LIN {X -0.145,Y -419.062,Z 861.894,A 0.000,B 0.000,C 90.000,E1 196.913} C_DIS
LIN {X 0.067,Y -417.772,Z 861.890,A 0.000,B 0.000,C 90.000,E1 196.205} C_DIS
LIN {X -0.189,Y -414.230,Z 861.881,A 0.000,B 0.000,C 90.000,E1 194.537} C_DIS
LIN {X -0.049,Y -408.722,Z 861.865,A 0.000,B 0.000,C 90.000,E1 191.771} C_DIS
LIN {X 0.119,Y -405.418,Z 861.856,A 0.000,B 0.000,C 90.000,E1 190.018} C_DIS
LIN {X 0.145,Y -402.699,Z 861.848,A 0.000,B 0.000,C 90.000,E1 188.624} C_DIS
LIN {X -0.116,Y -396.599,Z 861.831,A 0.000,B 0.000,C 90.000,E1 185.511} C_DIS
LIN {X -0.014,Y -390.296,Z 861.809,A 0.000,B 0.000,C 90.000,E1 181.604} C_DIS
LIN {X -0.149,Y -387.352,Z 861.797,A 0.000,B 0.000,C 90.000,E1 179.484} C_DIS
LIN {X 0.143,Y -384.816,Z 861.787,A 0.000,B 0.000,C 90.000,E1 177.650} C_DIS
LIN {X 0.018,Y -382.276,Z 861.777,A 0.000,B 0.000,C 90.000,E1 175.869} C_DIS
LIN {X 0.023,Y -378.755,Z 861.763,A 0.000,B 0.000,C 90.000,E1 173.337} C_DIS
LIN {X -0.169,Y -374.046,Z 861.739,A 0.000,B 0.000,C 90.000,E1 168.993} C_DIS
LIN {X -0.121,Y -373.099,Z 861.731,A 0.000,B 0.000,C 90.000,E1 167.521} C_DIS
LIN {X 0.156,Y -372.522,Z 861.720,A 0.000,B 0.000,C 90.000,E1 165.644} C_DIS
LIN {X -0.047,Y -372.718,Z 861.714,A 0.000,B 0.000,C 90.000,E1 164.574} C_DIS
LIN {X -0.080,Y -373.031,Z 861.712,A 0.000,B 0.000,C 90.000,E1 164.212} C_DIS
LIN {X -0.112,Y -373.157,Z 861.710,A 0.000,B 0.000,C 90.000,E1 163.850} C_DIS
LIN {X 0.127,Y -374.050,Z 861.705,A 0.000,B 0.000,C 90.000,E1 162.906} C_DIS
LIN {X 0.110,Y -375.461,Z 861.701,A 0.000,B 0.000,C 90.000,E1 162.127} C_DIS
LIN {X -0.174,Y -377.164,Z 861.698,A 0.000,B 0.000,C 90.000,E1 161.583} C_DIS
LIN {X -0.198,Y -379.423,Z 861.695,A 0.000,B 0.000,C 90.000,E1 161.040} C_DIS
LIN {X -0.203,Y -380.503,Z 861.694,A 0.000,B 0.000,C 90.000,E1 160.859} C_DIS
LIN {X -0.013,Y -383.679,Z 861.691,A 0.000,B 0.000,C 90.000,E1 160.369} C_DIS
LIN {X -0.012,Y -384.839,Z 861.690,A 0.000,B 0.000,C 90.000,E1 160.188} C_DIS
LIN {X -0.006,Y -386.584,Z 861.689,A 0.000,B 0.000,C 90.000,E1 160.007} C_DIS
LIN {X 0.011,Y -390.554,Z 861.687,A 0.000,B 0.000,C 90.000,E1 159.699} C_DIS
LIN {X 0.021,Y -392.446,Z 861.687,A 0.000,B 0.000,C 90.000,E1 159.571} C_DIS
LIN {X -0.042,Y -399.708,Z 861.685,A 0.000,B 0.000,C 90.000,E1 159.209} C_DIS
LIN {X -0.124,Y -407.378,Z 861.683,A 0.000,B 0.000,C 90.000,E1 158.901} C_DIS
LIN {X 0.178,Y -417.633,Z 861.680,A 0.000,B 0.000,C 90.000,E1 158.411} C_DIS
LIN {X -0.153,Y -425.580,Z 861.678,A 0.000,B 0.000,C 90.000,E1 158.028} C_DIS
LIN {X 0.034,Y -430.708,Z 861.676,A 0.000,B 0.000,C 90.000,E1 157.720} C_DIS
LIN {X -0.009,Y -433.655,Z 861.675,A 0.000,B 0.000,C 90.000,E1 157.539} C_DIS
LIN {X 0.068,Y -443.090,Z 861.672,A 0.000,B 0.000,C 90.000,E1 156.869} C_DIS
LIN {X -0.102,Y -447.734,Z 861.670,A 0.000,B 0.000,C 90.000,E1 156.538} C_DIS
LIN {X -0.139,Y -453.905,Z 861.667,A 0.000,B 0.000,C 90.000,E1 156.049} C_DIS
LIN {X -0.016,Y -464.227,Z 861.662,A 0.000,B 0.000,C 90.000,E1 155.101} C_DIS
LIN {X -0.106,Y -467.028,Z 861.660,A 0.000,B 0.000,C 90.000,E1 154.845} C_DIS
LIN {X -0.183,Y -472.623,Z 861.657,A 0.000,B 0.000,C 90.000,E1 154.280} C_DIS
LIN {X 0.095,Y -479.409,Z 861.653,A 0.000,B 0.000,C 90.000,E1 153.512} C_DIS
LIN {X 0.027,Y -483.253,Z 861.651,A 0.000,B 0.000,C 90.000,E1 153.076} C_DIS
LIN {X 0.252,Y -489.483,Z 861.646,A 0.000,B 0.000,C 90.000,E1 152.281} C_DIS
LIN {X 0.089,Y -495.170,Z 861.642,A 0.000,B 0.000,C 90.000,E1 151.591} C_DIS
LIN {X -0.181,Y -498.463,Z 861.640,A 0.000,B 0.000,C 90.000,E1 151.179} C_DIS
LIN {X -0.187,Y -503.200,Z 861.637,A 0.000,B 0.000,C 90.000,E1 150.589} C_DIS
LIN {X -0.265,Y -507.508,Z 861.633,A 0.000,B 0.000,C 90.000,E1 149.999} C_DIS
LIN {X -0.313,Y -511.672,Z 861.630,A 0.000,B 0.000,C 90.000,E1 149.410} C_DIS
LIN {X -0.155,Y -514.945,Z 861.627,A 0.000,B 0.000,C 90.000,E1 148.948} C_DIS
LIN {X 0.049,Y -520.575,Z 861.623,A 0.000,B 0.000,C 90.000,E1 148.043} C_DIS
LIN {X -0.231,Y -523.324,Z 861.620,A 0.000,B 0.000,C 90.000,E1 147.661} C_DIS
LIN {X -0.052,Y -527.781,Z 861.616,A 0.000,B 0.000,C 90.000,E1 146.914} C_DIS
LIN {X 0.019,Y -529.512,Z 861.615,A 0.000,B 0.000,C 90.000,E1 146.628} C_DIS
LIN {X 0.099,Y -536.054,Z 861.608,A 0.000,B 0.000,C 90.000,E1 145.468} C_DIS
LIN {X 0.120,Y -540.641,Z 861.604,A 0.000,B 0.000,C 90.000,E1 144.609} C_DIS
LIN {X -0.090,Y -546.662,Z 861.597,A 0.000,B 0.000,C 90.000,E1 143.497} C_DIS
LIN {X -0.202,Y -555.631,Z 861.588,A 0.000,B 0.000,C 90.000,E1 141.823} C_DIS
LIN {X -0.222,Y -563.196,Z 861.580,A 0.000,B 0.000,C 90.000,E1 140.436} C_DIS
LIN {X 0.135,Y -568.936,Z 861.574,A 0.000,B 0.000,C 90.000,E1 139.299} C_DIS
LIN {X -0.104,Y -573.699,Z 861.569,A 0.000,B 0.000,C 90.000,E1 138.366} C_DIS
LIN {X 0.017,Y -579.006,Z 861.563,A 0.000,B 0.000,C 90.000,E1 137.268} C_DIS
LIN {X 0.313,Y -585.693,Z 861.555,A 0.000,B 0.000,C 90.000,E1 135.891} C_DIS
LIN {X 0.022,Y -591.612,Z 861.548,A 0.000,B 0.000,C 90.000,E1 134.717} C_DIS
LIN {X -0.261,Y -595.300,Z 861.544,A 0.000,B 0.000,C 90.000,E1 133.947} C_DIS
LIN {X -0.093,Y -599.038,Z 861.540,A 0.000,B 0.000,C 90.000,E1 133.137} C_DIS
LIN {X -0.266,Y -605.015,Z 861.532,A 0.000,B 0.000,C 90.000,E1 131.838} C_DIS
LIN {X -0.150,Y -609.482,Z 861.527,A 0.000,B 0.000,C 90.000,E1 130.782} C_DIS
LIN {X -0.152,Y -614.771,Z 861.519,A 0.000,B 0.000,C 90.000,E1 129.483} C_DIS
LIN {X -0.294,Y -618.739,Z 861.514,A 0.000,B 0.000,C 90.000,E1 128.463} C_DIS
LIN {X -0.263,Y -625.196,Z 861.504,A 0.000,B 0.000,C 90.000,E1 126.664} C_DIS
LIN {X 0.239,Y -628.788,Z 861.498,A 0.000,B 0.000,C 90.000,E1 125.598} C_DIS
LIN {X -0.091,Y -631.992,Z 861.492,A 0.000,B 0.000,C 90.000,E1 124.612} C_DIS
LIN {X -0.242,Y -633.538,Z 861.490,A 0.000,B 0.000,C 90.000,E1 124.119} C_DIS
LIN {X 0.038,Y -636.798,Z 861.482,A 0.000,B 0.000,C 90.000,E1 122.832} C_DIS
LIN {X -0.046,Y -638.637,Z 861.478,A 0.000,B 0.000,C 90.000,E1 122.084} C_DIS
LIN {X 0.323,Y -641.263,Z 861.471,A 0.000,B 0.000,C 90.000,E1 120.797} C_DIS
LIN {X -0.157,Y -643.563,Z 861.464,A 0.000,B 0.000,C 90.000,E1 119.589} C_DIS
LIN {X -0.018,Y -644.146,Z 861.462,A 0.000,B 0.000,C 90.000,E1 119.077} C_DIS
LIN {X 0.130,Y -645.007,Z 861.459,A 0.000,B 0.000,C 90.000,E1 118.565} C_DIS
LIN {X -0.036,Y -646.885,Z 861.452,A 0.000,B 0.000,C 90.000,E1 117.334} C_DIS
LIN {X 0.136,Y -647.533,Z 861.449,A 0.000,B 0.000,C 90.000,E1 116.821} C_DIS
LIN {X 0.000,Y -648.671,Z 861.442,A 0.000,B 0.000,C 90.000,E1 115.591} C_DIS
LIN {X 0.090,Y -649.085,Z 861.437,A 0.000,B 0.000,C 90.000,E1 114.591} C_DIS
LIN {X 0.182,Y -649.129,Z 861.435,A 0.000,B 0.000,C 90.000,E1 114.335} C_DIS
LIN {X 0.363,Y -648.828,Z 861.433,A 0.000,B 0.000,C 90.000,E1 113.823} C_DIS
LIN {X 0.192,Y -648.419,Z 861.431,A 0.000,B 0.000,C 90.000,E1 113.590} C_DIS
LIN {X -0.229,Y -647.091,Z 861.428,A 0.000,B 0.000,C 90.000,E1 113.131} C_DIS
LIN {X -0.359,Y -644.836,Z 861.426,A 0.000,B 0.000,C 90.000,E1 112.770} C_DIS
LIN {X -0.320,Y -644.240,Z 861.426,A 0.000,B 0.000,C 90.000,E1 112.642} C_DIS
LIN {X -0.284,Y -643.376,Z 861.425,A 0.000,B 0.000,C 90.000,E1 112.514} C_DIS
LIN {X 0.377,Y -641.224,Z 861.424,A 0.000,B 0.000,C 90.000,E1 112.206} C_DIS
LIN {X 0.168,Y -640.004,Z 861.423,A 0.000,B 0.000,C 90.000,E1 112.099} C_DIS
LIN {X 0.207,Y -638.590,Z 861.422,A 0.000,B 0.000,C 90.000,E1 111.972} C_DIS
LIN {X 0.247,Y -636.605,Z 861.422,A 0.000,B 0.000,C 90.000,E1 111.844} C_DIS
LIN {X -0.279,Y -635.300,Z 861.421,A 0.000,B 0.000,C 90.000,E1 111.844} C_DIS
LIN {X -0.212,Y -631.962,Z 861.420,A 0.000,B 0.000,C 90.000,E1 111.589} C_DIS
LIN {X 0.146,Y -628.475,Z 861.419,A 0.000,B 0.000,C 90.000,E1 111.354} C_DIS
LIN {X -0.016,Y -623.661,Z 861.417,A 0.000,B 0.000,C 90.000,E1 111.099} C_DIS
LIN {X 0.310,Y -597.380,Z 861.410,A 0.000,B 0.000,C 90.000,E1 109.812} C_DIS
LIN {X 0.154,Y -589.216,Z 861.408,A 0.000,B 0.000,C 90.000,E1 109.450} C_DIS
LIN {X -0.233,Y -583.699,Z 861.407,A 0.000,B 0.000,C 90.000,E1 109.268} C_DIS
LIN {X 0.287,Y -580.083,Z 861.406,A 0.000,B 0.000,C 90.000,E1 109.087} C_DIS
LIN {X -0.189,Y -572.340,Z 861.405,A 0.000,B 0.000,C 90.000,E1 108.906} C_DIS
LIN {X 0.205,Y -566.390,Z 861.404,A 0.000,B 0.000,C 90.000,E1 108.671} C_DIS
LIN {X 0.035,Y -563.220,Z 861.403,A 0.000,B 0.000,C 90.000,E1 108.489} C_DIS
LIN {X -0.011,Y -562.426,Z 861.402,A 0.000,B 0.000,C 90.000,E1 108.417} C_DIS
LIN {X -0.223,Y -561.003,Z 861.401,A 0.000,B 0.000,C 90.000,E1 108.181} C_DIS
LIN {X -0.201,Y -559.978,Z 861.399,A 0.000,B 0.000,C 90.000,E1 107.764} C_DIS
LIN {X -0.142,Y -559.387,Z 861.395,A 0.000,B 0.000,C 90.000,E1 107.149} C_DIS
LIN {X 0.043,Y -559.497,Z 861.384,A 0.000,B 0.000,C 90.000,E1 105.190} C_DIS
LIN {X 0.130,Y -560.677,Z 861.369,A 0.000,B 0.000,C 90.000,E1 102.411} C_DIS
LIN {X 0.142,Y -562.134,Z 861.357,A 0.000,B 0.000,C 90.000,E1 100.197} C_DIS
LIN {X -0.122,Y -563.310,Z 861.348,A 0.000,B 0.000,C 90.000,E1 98.568} C_DIS
LIN {X -0.050,Y -564.232,Z 861.340,A 0.000,B 0.000,C 90.000,E1 97.182} C_DIS
LIN {X 0.038,Y -565.001,Z 861.332,A 0.000,B 0.000,C 90.000,E1 95.796} C_DIS
LIN {X -0.232,Y -565.860,Z 861.322,A 0.000,B 0.000,C 90.000,E1 93.898} C_DIS
LIN {X -0.213,Y -566.345,Z 861.314,A 0.000,B 0.000,C 90.000,E1 92.522} C_DIS
LIN {X -0.068,Y -566.780,Z 861.305,A 0.000,B 0.000,C 90.000,E1 90.859} C_DIS
LIN {X -0.042,Y -567.118,Z 861.297,A 0.000,B 0.000,C 90.000,E1 89.484} C_DIS
LIN {X 0.002,Y -567.427,Z 861.290,A 0.000,B 0.000,C 90.000,E1 88.108} C_DIS
LIN {X -0.278,Y -567.763,Z 861.279,A 0.000,B 0.000,C 90.000,E1 86.216} C_DIS
LIN {X -0.189,Y -567.981,Z 861.271,A 0.000,B 0.000,C 90.000,E1 84.837} C_DIS
LIN {X 0.240,Y -568.334,Z 861.261,A 0.000,B 0.000,C 90.000,E1 82.875} C_DIS
LIN {X -0.272,Y -568.959,Z 861.248,A 0.000,B 0.000,C 90.000,E1 80.735} C_DIS
LIN {X -0.027,Y -569.755,Z 861.236,A 0.000,B 0.000,C 90.000,E1 78.522} C_DIS
LIN {X 0.160,Y -570.549,Z 861.226,A 0.000,B 0.000,C 90.000,E1 76.589} C_DIS
LIN {X -0.066,Y -570.893,Z 861.220,A 0.000,B 0.000,C 90.000,E1 75.519} C_DIS
LIN {X 0.270,Y -571.198,Z 861.214,A 0.000,B 0.000,C 90.000,E1 74.393} C_DIS
LIN {X 0.057,Y -571.465,Z 861.207,A 0.000,B 0.000,C 90.000,E1 73.323} C_DIS
LIN {X 0.164,Y -571.700,Z 861.197,A 0.000,B 0.000,C 90.000,E1 71.402} C_DIS
LIN {X -0.087,Y -571.730,Z 861.186,A 0.000,B 0.000,C 90.000,E1 69.518} C_DIS
LIN {X 0.249,Y -571.730,Z 861.177,A 0.000,B 0.000,C 90.000,E1 67.847} C_DIS
LIN {X 0.063,Y -571.623,Z 861.168,A 0.000,B 0.000,C 90.000,E1 66.230} C_DIS
LIN {X 0.270,Y -571.464,Z 861.160,A 0.000,B 0.000,C 90.000,E1 64.845} C_DIS
LIN {X -0.212,Y -571.079,Z 861.151,A 0.000,B 0.000,C 90.000,E1 63.256} C_DIS
LIN {X 0.054,Y -570.536,Z 861.142,A 0.000,B 0.000,C 90.000,E1 61.591} C_DIS
LIN {X -0.078,Y -570.026,Z 861.136,A 0.000,B 0.000,C 90.000,E1 60.511} C_DIS
LIN {X 0.179,Y -569.623,Z 861.132,A 0.000,B 0.000,C 90.000,E1 59.665} C_DIS
LIN {X -0.133,Y -568.550,Z 861.124,A 0.000,B 0.000,C 90.000,E1 58.329} C_DIS
LIN {X -0.088,Y -567.894,Z 861.119,A 0.000,B 0.000,C 90.000,E1 57.502} C_DIS
LIN {X -0.356,Y -567.033,Z 861.115,A 0.000,B 0.000,C 90.000,E1 56.707} C_DIS
LIN {X -0.213,Y -565.644,Z 861.109,A 0.000,B 0.000,C 90.000,E1 55.595} C_DIS
LIN {X -0.199,Y -564.517,Z 861.104,A 0.000,B 0.000,C 90.000,E1 54.769} C_DIS
LIN {X 0.234,Y -562.850,Z 861.098,A 0.000,B 0.000,C 90.000,E1 53.623} C_DIS
LIN {X -0.141,Y -560.884,Z 861.092,A 0.000,B 0.000,C 90.000,E1 52.557} C_DIS
LIN {X 0.145,Y -559.235,Z 861.087,A 0.000,B 0.000,C 90.000,E1 51.698} C_DIS
LIN {X -0.113,Y -558.053,Z 861.084,A 0.000,B 0.000,C 90.000,E1 51.170} C_DIS
LIN {X -0.294,Y -555.992,Z 861.080,A 0.000,B 0.000,C 90.000,E1 50.356} C_DIS
LIN {X 0.284,Y -553.563,Z 861.075,A 0.000,B 0.000,C 90.000,E1 49.461} C_DIS
LIN {X 0.050,Y -550.841,Z 861.070,A 0.000,B 0.000,C 90.000,E1 48.647} C_DIS
LIN {X 0.106,Y -548.875,Z 861.067,A 0.000,B 0.000,C 90.000,E1 48.081} C_DIS
LIN {X 0.187,Y -545.568,Z 861.063,A 0.000,B 0.000,C 90.000,E1 47.229} C_DIS
LIN {X 0.036,Y -542.567,Z 861.059,A 0.000,B 0.000,C 90.000,E1 46.539} C_DIS
LIN {X 0.228,Y -539.269,Z 861.055,A 0.000,B 0.000,C 90.000,E1 45.810} C_DIS
LIN {X 0.022,Y -537.203,Z 861.052,A 0.000,B 0.000,C 90.000,E1 45.405} C_DIS
LIN {X 0.165,Y -533.249,Z 861.048,A 0.000,B 0.000,C 90.000,E1 44.676} C_DIS
LIN {X 0.101,Y -529.791,Z 861.045,A 0.000,B 0.000,C 90.000,E1 44.109} C_DIS
LIN {X 0.077,Y -526.153,Z 861.042,A 0.000,B 0.000,C 90.000,E1 43.542} C_DIS
LIN {X -0.042,Y -522.226,Z 861.039,A 0.000,B 0.000,C 90.000,E1 42.975} C_DIS
LIN {X 0.193,Y -517.988,Z 861.036,A 0.000,B 0.000,C 90.000,E1 42.366} C_DIS
LIN {X -0.331,Y -513.435,Z 861.032,A 0.000,B 0.000,C 90.000,E1 41.838} C_DIS
LIN {X 0.055,Y -509.906,Z 861.030,A 0.000,B 0.000,C 90.000,E1 41.353} C_DIS
LIN {X 0.067,Y -504.988,Z 861.027,A 0.000,B 0.000,C 90.000,E1 40.782} C_DIS
LIN {X -0.141,Y -500.047,Z 861.024,A 0.000,B 0.000,C 90.000,E1 40.253} C_DIS
LIN {X -0.038,Y -495.889,Z 861.021,A 0.000,B 0.000,C 90.000,E1 39.806} C_DIS
LIN {X -0.212,Y -490.304,Z 861.018,A 0.000,B 0.000,C 90.000,E1 39.277} C_DIS
LIN {X -0.153,Y -481.649,Z 861.014,A 0.000,B 0.000,C 90.000,E1 38.463} C_DIS
LIN {X 0.113,Y -470.949,Z 861.009,A 0.000,B 0.000,C 90.000,E1 37.523} C_DIS
LIN {X 0.015,Y -464.758,Z 861.006,A 0.000,B 0.000,C 90.000,E1 37.030} C_DIS
LIN {X -0.286,Y -452.263,Z 861.000,A 0.000,B 0.000,C 90.000,E1 36.091} C_DIS
LIN {X 0.081,Y -438.081,Z 860.994,A 0.000,B 0.000,C 90.000,E1 34.945} C_DIS
LIN {X 0.012,Y -419.665,Z 860.986,A 0.000,B 0.000,C 90.000,E1 33.452} C_DIS
LIN {X 0.029,Y -404.695,Z 860.978,A 0.000,B 0.000,C 90.000,E1 32.084} C_DIS
LIN {X -0.041,Y -399.160,Z 860.975,A 0.000,B 0.000,C 90.000,E1 31.514} C_DIS
LIN {X -0.019,Y -394.767,Z 860.972,A 0.000,B 0.000,C 90.000,E1 30.924} C_DIS
LIN {X 0.013,Y -393.080,Z 860.970,A 0.000,B 0.000,C 90.000,E1 30.590} C_DIS
LIN {X 0.017,Y -392.132,Z 860.969,A 0.000,B 0.000,C 90.000,E1 30.413} C_DIS
LIN {X -0.239,Y -390.569,Z 860.966,A 0.000,B 0.000,C 90.000,E1 29.873} C_DIS
LIN {X -0.005,Y -389.839,Z 860.961,A 0.000,B 0.000,C 90.000,E1 28.949} C_DIS
LIN {X 0.031,Y -389.754,Z 860.957,A 0.000,B 0.000,C 90.000,E1 28.231} C_DIS
LIN {X -0.106,Y -392.270,Z 860.935,A 0.000,B 0.000,C 90.000,E1 24.335} C_DIS
LIN {X 0.208,Y -395.035,Z 860.917,A 0.000,B 0.000,C 90.000,E1 21.099} C_DIS
LIN {X -0.081,Y -397.526,Z 860.904,A 0.000,B 0.000,C 90.000,E1 18.671} C_DIS
LIN {X -0.087,Y -399.530,Z 860.894,A 0.000,B 0.000,C 90.000,E1 16.913} C_DIS
LIN {X -0.136,Y -403.103,Z 860.878,A 0.000,B 0.000,C 90.000,E1 14.120} C_DIS
LIN {X 0.129,Y -407.132,Z 860.863,A 0.000,B 0.000,C 90.000,E1 11.299} C_DIS
LIN {X -0.138,Y -410.967,Z 860.849,A 0.000,B 0.000,C 90.000,E1 8.916} C_DIS
LIN {X 0.088,Y -416.322,Z 860.832,A 0.000,B 0.000,C 90.000,E1 5.796} C_DIS
LIN {X -0.144,Y -420.094,Z 860.821,A 0.000,B 0.000,C 90.000,E1 3.784} C_DIS
LIN {X 0.203,Y -425.720,Z 860.806,A 0.000,B 0.000,C 90.000,E1 1.031} C_DIS
LIN {X -0.199,Y -429.433,Z 860.797,A 0.000,B 0.000,C 90.000,E1 359.484} C_DIS
LIN {X -0.076,Y -435.036,Z 860.784,A 0.000,B 0.000,C 90.000,E1 357.135} C_DIS
LIN {X -0.040,Y -441.939,Z 860.769,A 0.000,B 0.000,C 90.000,E1 354.489} C_DIS
LIN {X -0.159,Y -444.717,Z 860.765,A 0.000,B 0.000,C 90.000,E1 353.685} C_DIS
LIN {X -0.185,Y -446.635,Z 860.763,A 0.000,B 0.000,C 90.000,E1 353.280} C_DIS
LIN {X -0.205,Y -451.971,Z 860.759,A 0.000,B 0.000,C 90.000,E1 352.648} C_DIS
LIN {X -0.058,Y -455.920,Z 860.758,A 0.000,B 0.000,C 90.000,E1 352.356} C_DIS
LIN {X 0.064,Y -462.281,Z 860.756,A 0.000,B 0.000,C 90.000,E1 352.008} C_DIS
LIN {X -0.177,Y -473.870,Z 860.753,A 0.000,B 0.000,C 90.000,E1 351.489} C_DIS
LIN {X -0.152,Y -480.634,Z 860.751,A 0.000,B 0.000,C 90.000,E1 351.141} C_DIS
LIN {X 0.231,Y -486.952,Z 860.749,A 0.000,B 0.000,C 90.000,E1 350.735} C_DIS
LIN {X 0.226,Y -496.803,Z 860.745,A 0.000,B 0.000,C 90.000,E1 350.151} C_DIS
LIN {X 0.094,Y -507.807,Z 860.742,A 0.000,B 0.000,C 90.000,E1 349.454} C_DIS
LIN {X 0.192,Y -517.208,Z 860.738,A 0.000,B 0.000,C 90.000,E1 348.814} C_DIS
LIN {X 0.075,Y -526.384,Z 860.734,A 0.000,B 0.000,C 90.000,E1 348.173} C_DIS
LIN {X -0.235,Y -533.792,Z 860.731,A 0.000,B 0.000,C 90.000,E1 347.645} C_DIS
LIN {X -0.178,Y -541.052,Z 860.728,A 0.000,B 0.000,C 90.000,E1 347.048} C_DIS
LIN {X 0.009,Y -550.870,Z 860.723,A 0.000,B 0.000,C 90.000,E1 346.172} C_DIS
LIN {X -0.115,Y -560.007,Z 860.718,A 0.000,B 0.000,C 90.000,E1 345.283} C_DIS
LIN {X -0.172,Y -565.040,Z 860.715,A 0.000,B 0.000,C 90.000,E1 344.755} C_DIS
LIN {X 0.126,Y -572.253,Z 860.711,A 0.000,B 0.000,C 90.000,E1 343.921} C_DIS
LIN {X -0.148,Y -577.732,Z 860.707,A 0.000,B 0.000,C 90.000,E1 343.268} C_DIS
LIN {X 0.259,Y -583.987,Z 860.703,A 0.000,B 0.000,C 90.000,E1 342.417} C_DIS
LIN {X 0.146,Y -587.838,Z 860.700,A 0.000,B 0.000,C 90.000,E1 341.891} C_DIS
LIN {X 0.174,Y -592.324,Z 860.696,A 0.000,B 0.000,C 90.000,E1 341.221} C_DIS
LIN {X 0.189,Y -597.396,Z 860.691,A 0.000,B 0.000,C 90.000,E1 340.423} C_DIS
LIN {X 0.009,Y -602.864,Z 860.686,A 0.000,B 0.000,C 90.000,E1 339.518} C_DIS
LIN {X 0.047,Y -609.460,Z 860.680,A 0.000,B 0.000,C 90.000,E1 338.337} C_DIS
LIN {X 0.227,Y -614.416,Z 860.675,A 0.000,B 0.000,C 90.000,E1 337.411} C_DIS
LIN {X -0.111,Y -619.731,Z 860.669,A 0.000,B 0.000,C 90.000,E1 336.410} C_DIS
LIN {X 0.184,Y -623.516,Z 860.665,A 0.000,B 0.000,C 90.000,E1 335.613} C_DIS
LIN {X 0.233,Y -629.342,Z 860.658,A 0.000,B 0.000,C 90.000,E1 334.332} C_DIS
LIN {X 0.034,Y -632.552,Z 860.653,A 0.000,B 0.000,C 90.000,E1 333.589} C_DIS
LIN {X 0.141,Y -635.611,Z 860.649,A 0.000,B 0.000,C 90.000,E1 332.820} C_DIS
LIN {X -0.236,Y -639.523,Z 860.644,A 0.000,B 0.000,C 90.000,E1 331.847} C_DIS
LIN {X 0.310,Y -643.100,Z 860.638,A 0.000,B 0.000,C 90.000,E1 330.795} C_DIS
LIN {X 0.353,Y -646.615,Z 860.632,A 0.000,B 0.000,C 90.000,E1 329.793} C_DIS
LIN {X 0.030,Y -649.075,Z 860.628,A 0.000,B 0.000,C 90.000,E1 329.076} C_DIS
LIN {X -0.318,Y -652.863,Z 860.621,A 0.000,B 0.000,C 90.000,E1 327.867} C_DIS
LIN {X 0.201,Y -655.609,Z 860.616,A 0.000,B 0.000,C 90.000,E1 326.834} C_DIS
LIN {X 0.299,Y -657.575,Z 860.612,A 0.000,B 0.000,C 90.000,E1 326.087} C_DIS
LIN {X -0.100,Y -660.554,Z 860.605,A 0.000,B 0.000,C 90.000,E1 324.895} C_DIS
LIN {X -0.016,Y -662.610,Z 860.600,A 0.000,B 0.000,C 90.000,E1 323.909} C_DIS
LIN {X 0.092,Y -664.473,Z 860.594,A 0.000,B 0.000,C 90.000,E1 322.924} C_DIS
LIN {X 0.189,Y -666.414,Z 860.587,A 0.000,B 0.000,C 90.000,E1 321.698} C_DIS
LIN {X -0.205,Y -668.169,Z 860.581,A 0.000,B 0.000,C 90.000,E1 320.517} C_DIS
LIN {X 0.291,Y -669.078,Z 860.577,A 0.000,B 0.000,C 90.000,E1 319.747} C_DIS
LIN {X -0.061,Y -670.675,Z 860.568,A 0.000,B 0.000,C 90.000,E1 318.324} C_DIS
LIN {X 0.088,Y -672.973,Z 860.558,A 0.000,B 0.000,C 90.000,E1 316.377} C_DIS
LIN {X 0.201,Y -674.442,Z 860.551,A 0.000,B 0.000,C 90.000,E1 315.162} C_DIS
LIN {X 0.226,Y -674.593,Z 860.550,A 0.000,B 0.000,C 90.000,E1 314.919} C_DIS
LIN {X 0.253,Y -674.941,Z 860.548,A 0.000,B 0.000,C 90.000,E1 314.676} C_DIS
LIN {X 0.054,Y -677.032,Z 860.536,A 0.000,B 0.000,C 90.000,E1 312.528} C_DIS
LIN {X 0.265,Y -678.191,Z 860.530,A 0.000,B 0.000,C 90.000,E1 311.310} C_DIS
LIN {X 0.121,Y -679.752,Z 860.520,A 0.000,B 0.000,C 90.000,E1 309.644} C_DIS
LIN {X -0.091,Y -680.568,Z 860.515,A 0.000,B 0.000,C 90.000,E1 308.705} C_DIS
LIN {X -0.083,Y -681.939,Z 860.506,A 0.000,B 0.000,C 90.000,E1 307.030} C_DIS
LIN {X -0.078,Y -683.066,Z 860.498,A 0.000,B 0.000,C 90.000,E1 305.598} C_DIS
LIN {X -0.457,Y -684.012,Z 860.490,A 0.000,B 0.000,C 90.000,E1 304.199} C_DIS
LIN {X -0.060,Y -685.313,Z 860.479,A 0.000,B 0.000,C 90.000,E1 302.260} C_DIS
LIN {X 0.003,Y -686.563,Z 860.470,A 0.000,B 0.000,C 90.000,E1 300.590} C_DIS
LIN {X -0.245,Y -687.943,Z 860.461,A 0.000,B 0.000,C 90.000,E1 298.949} C_DIS
LIN {X -0.087,Y -689.285,Z 860.453,A 0.000,B 0.000,C 90.000,E1 297.513} C_DIS
LIN {X 0.016,Y -690.960,Z 860.444,A 0.000,B 0.000,C 90.000,E1 295.848} C_DIS
LIN {X 0.292,Y -692.132,Z 860.437,A 0.000,B 0.000,C 90.000,E1 294.643} C_DIS
LIN {X 0.099,Y -692.644,Z 860.433,A 0.000,B 0.000,C 90.000,E1 293.951} C_DIS
LIN {X -0.092,Y -692.634,Z 860.429,A 0.000,B 0.000,C 90.000,E1 293.259} C_DIS
LIN {X 0.114,Y -691.666,Z 860.427,A 0.000,B 0.000,C 90.000,E1 292.770} C_DIS
LIN {X 0.351,Y -690.965,Z 860.425,A 0.000,B 0.000,C 90.000,E1 292.514} C_DIS
LIN {X 0.203,Y -690.295,Z 860.425,A 0.000,B 0.000,C 90.000,E1 292.408} C_DIS
LIN {X -0.238,Y -686.592,Z 860.422,A 0.000,B 0.000,C 90.000,E1 291.972} C_DIS
LIN {X -0.127,Y -685.449,Z 860.421,A 0.000,B 0.000,C 90.000,E1 291.844} C_DIS
LIN {X -0.021,Y -683.688,Z 860.421,A 0.000,B 0.000,C 90.000,E1 291.716} C_DIS
LIN {X -0.179,Y -679.497,Z 860.420,A 0.000,B 0.000,C 90.000,E1 291.535} C_DIS
LIN {X 0.264,Y -676.010,Z 860.419,A 0.000,B 0.000,C 90.000,E1 291.354} C_DIS
LIN {X 0.166,Y -670.319,Z 860.418,A 0.000,B 0.000,C 90.000,E1 291.173} C_DIS
LIN {X 0.140,Y -656.825,Z 860.416,A 0.000,B 0.000,C 90.000,E1 290.865} C_DIS
LIN {X -0.130,Y -653.809,Z 860.415,A 0.000,B 0.000,C 90.000,E1 290.791} C_DIS
LIN {X -0.178,Y -648.988,Z 860.414,A 0.000,B 0.000,C 90.000,E1 290.610} C_DIS
LIN {X 0.109,Y -645.497,Z 860.413,A 0.000,B 0.000,C 90.000,E1 290.375} C_DIS
LIN {X 0.075,Y -645.452,Z 860.413,A 0.000,B 0.000,C 90.000,E1 290.375} C_DIS
LIN {X 0.063,Y -644.354,Z 860.412,A 0.000,B 0.000,C 90.000,E1 290.194} C_DIS
LIN {X 0.242,Y -644.350,Z 860.412,A 0.000,B 0.000,C 90.000,E1 290.174} C_DIS
LIN {X 0.299,Y -644.577,Z 860.411,A 0.000,B 0.000,C 90.000,E1 289.939} C_DIS
LIN {X 0.168,Y -646.105,Z 860.409,A 0.000,B 0.000,C 90.000,E1 289.577} C_DIS
LIN {X 0.145,Y -648.591,Z 860.406,A 0.000,B 0.000,C 90.000,E1 289.087} C_DIS
LIN {X -0.205,Y -653.932,Z 860.401,A 0.000,B 0.000,C 90.000,E1 288.127} C_DIS
LIN {X -0.375,Y -657.446,Z 860.397,A 0.000,B 0.000,C 90.000,E1 287.402} C_DIS
LIN {X 0.115,Y -660.564,Z 860.392,A 0.000,B 0.000,C 90.000,E1 286.622} C_DIS
LIN {X 0.097,Y -662.428,Z 860.390,A 0.000,B 0.000,C 90.000,E1 286.134} C_DIS
LIN {X -0.184,Y -664.701,Z 860.386,A 0.000,B 0.000,C 90.000,E1 285.426} C_DIS
LIN {X -0.358,Y -666.004,Z 860.383,A 0.000,B 0.000,C 90.000,E1 284.954} C_DIS
LIN {X 0.047,Y -667.542,Z 860.379,A 0.000,B 0.000,C 90.000,E1 284.189} C_DIS
LIN {X 0.055,Y -668.351,Z 860.376,A 0.000,B 0.000,C 90.000,E1 283.703} C_DIS
LIN {X -0.321,Y -669.167,Z 860.372,A 0.000,B 0.000,C 90.000,E1 283.008} C_DIS
LIN {X 0.049,Y -669.893,Z 860.367,A 0.000,B 0.000,C 90.000,E1 282.007} C_DIS
LIN {X -0.093,Y -669.949,Z 860.364,A 0.000,B 0.000,C 90.000,E1 281.535} C_DIS
LIN {X 0.219,Y -669.577,Z 860.360,A 0.000,B 0.000,C 90.000,E1 280.782} C_DIS
LIN {X 0.071,Y -669.107,Z 860.357,A 0.000,B 0.000,C 90.000,E1 280.310} C_DIS
LIN {X -0.200,Y -668.361,Z 860.355,A 0.000,B 0.000,C 90.000,E1 279.849} C_DIS
LIN {X 0.297,Y -667.316,Z 860.352,A 0.000,B 0.000,C 90.000,E1 279.321} C_DIS
LIN {X 0.019,Y -665.999,Z 860.349,A 0.000,B 0.000,C 90.000,E1 278.859} C_DIS
LIN {X -0.071,Y -665.235,Z 860.348,A 0.000,B 0.000,C 90.000,E1 278.624} C_DIS
LIN {X 0.298,Y -663.415,Z 860.345,A 0.000,B 0.000,C 90.000,E1 278.106} C_DIS
LIN {X 0.001,Y -661.228,Z 860.343,A 0.000,B 0.000,C 90.000,E1 277.644} C_DIS
LIN {X 0.247,Y -658.110,Z 860.339,A 0.000,B 0.000,C 90.000,E1 277.011} C_DIS
LIN {X -0.110,Y -654.335,Z 860.336,A 0.000,B 0.000,C 90.000,E1 276.429} C_DIS
LIN {X 0.222,Y -651.852,Z 860.334,A 0.000,B 0.000,C 90.000,E1 276.030} C_DIS
LIN {X -0.195,Y -646.896,Z 860.330,A 0.000,B 0.000,C 90.000,E1 275.448} C_DIS
LIN {X -0.006,Y -642.240,Z 860.327,A 0.000,B 0.000,C 90.000,E1 274.935} C_DIS
LIN {X -0.282,Y -637.000,Z 860.325,A 0.000,B 0.000,C 90.000,E1 274.473} C_DIS
LIN {X 0.022,Y -631.855,Z 860.322,A 0.000,B 0.000,C 90.000,E1 274.012} C_DIS
LIN {X -0.225,Y -624.567,Z 860.319,A 0.000,B 0.000,C 90.000,E1 273.498} C_DIS
LIN {X 0.099,Y -616.864,Z 860.317,A 0.000,B 0.000,C 90.000,E1 272.980} C_DIS
LIN {X -0.157,Y -610.418,Z 860.315,A 0.000,B 0.000,C 90.000,E1 272.636} C_DIS
LIN {X -0.071,Y -603.467,Z 860.313,A 0.000,B 0.000,C 90.000,E1 272.293} C_DIS
LIN {X -0.242,Y -596.376,Z 860.311,A 0.000,B 0.000,C 90.000,E1 272.007} C_DIS
LIN {X 0.114,Y -590.742,Z 860.310,A 0.000,B 0.000,C 90.000,E1 271.776} C_DIS
LIN {X 0.233,Y -583.324,Z 860.309,A 0.000,B 0.000,C 90.000,E1 271.547} C_DIS
LIN {X 0.032,Y -577.629,Z 860.308,A 0.000,B 0.000,C 90.000,E1 271.432} C_DIS
LIN {X 0.054,Y -569.923,Z 860.307,A 0.000,B 0.000,C 90.000,E1 271.318} C_DIS
LIN {X 0.166,Y -564.443,Z 860.307,A 0.000,B 0.000,C 90.000,E1 271.260} C_DIS
LIN {X -0.264,Y -554.469,Z 860.307,A 0.000,B 0.000,C 90.000,E1 271.260} C_DIS
LIN {X -0.019,Y -552.014,Z 860.307,A 0.000,B 0.000,C 90.000,E1 271.203} C_DIS
LIN {X -0.006,Y -550.118,Z 860.306,A 0.000,B 0.000,C 90.000,E1 271.146} C_DIS
LIN {X -0.037,Y -550.079,Z 860.306,A 0.000,B 0.000,C 90.000,E1 271.146} C_DIS
LIN {X -0.060,Y -547.855,Z 860.305,A 0.000,B 0.000,C 90.000,E1 270.859} C_DIS
LIN {X -0.015,Y -547.374,Z 860.305,A 0.000,B 0.000,C 90.000,E1 270.802} C_DIS
LIN {X -0.058,Y -547.340,Z 860.304,A 0.000,B 0.000,C 90.000,E1 270.802} C_DIS
LIN {X -0.091,Y -546.335,Z 860.301,A 0.000,B 0.000,C 90.000,E1 270.229} C_DIS
LIN {X -0.205,Y -543.573,Z 860.284,A 0.000,B 0.000,C 90.000,E1 267.135} C_DIS
LIN {X 0.017,Y -542.467,Z 860.275,A 0.000,B 0.000,C 90.000,E1 265.412} C_DIS
LIN {X 0.260,Y -541.253,Z 860.265,A 0.000,B 0.000,C 90.000,E1 263.685} C_DIS
LIN {X -0.133,Y -540.285,Z 860.259,A 0.000,B 0.000,C 90.000,E1 262.591} C_DIS
LIN {X -0.002,Y -539.508,Z 860.254,A 0.000,B 0.000,C 90.000,E1 261.724} C_DIS
LIN {X -0.216,Y -537.977,Z 860.245,A 0.000,B 0.000,C 90.000,E1 260.038} C_DIS
LIN {X 0.105,Y -536.542,Z 860.237,A 0.000,B 0.000,C 90.000,E1 258.578} C_DIS
LIN {X -0.124,Y -535.021,Z 860.229,A 0.000,B 0.000,C 90.000,E1 257.173} C_DIS
LIN {X 0.257,Y -533.290,Z 860.221,A 0.000,B 0.000,C 90.000,E1 255.700} C_DIS
LIN {X -0.038,Y -530.491,Z 860.208,A 0.000,B 0.000,C 90.000,E1 253.433} C_DIS
LIN {X 0.063,Y -528.484,Z 860.198,A 0.000,B 0.000,C 90.000,E1 251.692} C_DIS
LIN {X -0.069,Y -526.973,Z 860.192,A 0.000,B 0.000,C 90.000,E1 250.550} C_DIS
LIN {X -0.226,Y -524.286,Z 860.181,A 0.000,B 0.000,C 90.000,E1 248.539} C_DIS
LIN {X -0.223,Y -521.693,Z 860.171,A 0.000,B 0.000,C 90.000,E1 246.794} C_DIS
LIN {X 0.052,Y -519.443,Z 860.163,A 0.000,B 0.000,C 90.000,E1 245.305} C_DIS
LIN {X 0.021,Y -517.229,Z 860.155,A 0.000,B 0.000,C 90.000,E1 243.845} C_DIS
LIN {X -0.161,Y -514.126,Z 860.145,A 0.000,B 0.000,C 90.000,E1 242.103} C_DIS
LIN {X -0.164,Y -511.121,Z 860.135,A 0.000,B 0.000,C 90.000,E1 240.333} C_DIS
LIN {X 0.019,Y -507.766,Z 860.125,A 0.000,B 0.000,C 90.000,E1 238.535} C_DIS
LIN {X 0.076,Y -504.867,Z 860.117,A 0.000,B 0.000,C 90.000,E1 237.041} C_DIS
LIN {X -0.227,Y -502.443,Z 860.110,A 0.000,B 0.000,C 90.000,E1 235.881} C_DIS
LIN {X -0.164,Y -500.498,Z 860.105,A 0.000,B 0.000,C 90.000,E1 234.975} C_DIS
LIN {X -0.124,Y -498.392,Z 860.100,A 0.000,B 0.000,C 90.000,E1 234.069} C_DIS
LIN {X -0.062,Y -493.330,Z 860.089,A 0.000,B 0.000,C 90.000,E1 231.949} C_DIS
LIN {X -0.122,Y -488.381,Z 860.077,A 0.000,B 0.000,C 90.000,E1 229.828} C_DIS
LIN {X -0.309,Y -486.240,Z 860.072,A 0.000,B 0.000,C 90.000,E1 228.933} C_DIS
LIN {X -0.176,Y -480.805,Z 860.058,A 0.000,B 0.000,C 90.000,E1 226.458} C_DIS
LIN {X -0.005,Y -476.165,Z 860.046,A 0.000,B 0.000,C 90.000,E1 224.271} C_DIS
LIN {X 0.189,Y -472.793,Z 860.037,A 0.000,B 0.000,C 90.000,E1 222.690} C_DIS
LIN {X 0.072,Y -468.696,Z 860.027,A 0.000,B 0.000,C 90.000,E1 220.825} C_DIS
LIN {X -0.094,Y -464.676,Z 860.016,A 0.000,B 0.000,C 90.000,E1 218.955} C_DIS
LIN {X -0.057,Y -462.034,Z 860.009,A 0.000,B 0.000,C 90.000,E1 217.684} C_DIS
LIN {X -0.032,Y -458.734,Z 860.001,A 0.000,B 0.000,C 90.000,E1 216.091} C_DIS
LIN {X 0.106,Y -453.883,Z 859.988,A 0.000,B 0.000,C 90.000,E1 213.833} C_DIS
LIN {X -0.104,Y -449.763,Z 859.977,A 0.000,B 0.000,C 90.000,E1 211.926} C_DIS
LIN {X -0.256,Y -445.544,Z 859.967,A 0.000,B 0.000,C 90.000,E1 210.001} C_DIS
LIN {X -0.169,Y -442.251,Z 859.957,A 0.000,B 0.000,C 90.000,E1 208.359} C_DIS
LIN {X 0.036,Y -438.852,Z 859.948,A 0.000,B 0.000,C 90.000,E1 206.693} C_DIS
LIN {X 0.009,Y -434.052,Z 859.936,A 0.000,B 0.000,C 90.000,E1 204.387} C_DIS
LIN {X 0.083,Y -430.622,Z 859.926,A 0.000,B 0.000,C 90.000,E1 202.717} C_DIS
LIN {X 0.096,Y -427.263,Z 859.917,A 0.000,B 0.000,C 90.000,E1 201.046} C_DIS
LIN {X -0.112,Y -423.989,Z 859.908,A 0.000,B 0.000,C 90.000,E1 199.396} C_DIS
LIN {X 0.058,Y -420.056,Z 859.896,A 0.000,B 0.000,C 90.000,E1 197.347} C_DIS
LIN {X 0.165,Y -418.169,Z 859.891,A 0.000,B 0.000,C 90.000,E1 196.315} C_DIS
LIN {X -0.091,Y -414.604,Z 859.881,A 0.000,B 0.000,C 90.000,E1 194.647} C_DIS
LIN {X -0.089,Y -410.380,Z 859.870,A 0.000,B 0.000,C 90.000,E1 192.591} C_DIS
LIN {X 0.096,Y -407.756,Z 859.862,A 0.000,B 0.000,C 90.000,E1 191.186} C_DIS
LIN {X 0.163,Y -405.133,Z 859.855,A 0.000,B 0.000,C 90.000,E1 189.792} C_DIS
LIN {X 0.188,Y -401.680,Z 859.845,A 0.000,B 0.000,C 90.000,E1 188.049} C_DIS
LIN {X -0.035,Y -396.291,Z 859.829,A 0.000,B 0.000,C 90.000,E1 185.277} C_DIS
LIN {X -0.060,Y -392.206,Z 859.816,A 0.000,B 0.000,C 90.000,E1 182.808} C_DIS
LIN {X 0.159,Y -388.666,Z 859.802,A 0.000,B 0.000,C 90.000,E1 180.286} C_DIS
LIN {X 0.082,Y -386.190,Z 859.792,A 0.000,B 0.000,C 90.000,E1 178.511} C_DIS
LIN {X -0.133,Y -383.139,Z 859.780,A 0.000,B 0.000,C 90.000,E1 176.388} C_DIS
LIN {X -0.169,Y -381.091,Z 859.772,A 0.000,B 0.000,C 90.000,E1 174.951} C_DIS
LIN {X 0.117,Y -377.326,Z 859.756,A 0.000,B 0.000,C 90.000,E1 172.008} C_DIS
LIN {X 0.106,Y -373.487,Z 859.733,A 0.000,B 0.000,C 90.000,E1 167.993} C_DIS
LIN {X -0.139,Y -372.326,Z 859.719,A 0.000,B 0.000,C 90.000,E1 165.463} C_DIS
LIN {X -0.017,Y -372.634,Z 859.711,A 0.000,B 0.000,C 90.000,E1 163.976} C_DIS
LIN {X -0.172,Y -373.382,Z 859.705,A 0.000,B 0.000,C 90.000,E1 162.906} C_DIS
LIN {X -0.201,Y -374.049,Z 859.703,A 0.000,B 0.000,C 90.000,E1 162.543} C_DIS
LIN {X 0.127,Y -374.514,Z 859.701,A 0.000,B 0.000,C 90.000,E1 162.127} C_DIS
LIN {X 0.102,Y -375.433,Z 859.699,A 0.000,B 0.000,C 90.000,E1 161.764} C_DIS
LIN {X 0.071,Y -376.543,Z 859.696,A 0.000,B 0.000,C 90.000,E1 161.221} C_DIS
LIN {X 0.036,Y -377.884,Z 859.694,A 0.000,B 0.000,C 90.000,E1 160.859} C_DIS
LIN {X 0.023,Y -379.353,Z 859.692,A 0.000,B 0.000,C 90.000,E1 160.496} C_DIS
LIN {X -0.130,Y -381.076,Z 859.690,A 0.000,B 0.000,C 90.000,E1 160.188} C_DIS
LIN {X -0.005,Y -382.121,Z 859.689,A 0.000,B 0.000,C 90.000,E1 160.007} C_DIS
LIN {X -0.041,Y -386.412,Z 859.686,A 0.000,B 0.000,C 90.000,E1 159.518} C_DIS
LIN {X 0.035,Y -388.364,Z 859.685,A 0.000,B 0.000,C 90.000,E1 159.337} C_DIS
LIN {X 0.001,Y -394.442,Z 859.683,A 0.000,B 0.000,C 90.000,E1 158.954} C_DIS
LIN {X 0.131,Y -401.521,Z 859.681,A 0.000,B 0.000,C 90.000,E1 158.592} C_DIS
LIN {X 0.176,Y -412.181,Z 859.679,A 0.000,B 0.000,C 90.000,E1 158.156} C_DIS
LIN {X 0.056,Y -415.535,Z 859.678,A 0.000,B 0.000,C 90.000,E1 158.028} C_DIS
LIN {X -0.045,Y -421.913,Z 859.676,A 0.000,B 0.000,C 90.000,E1 157.720} C_DIS
LIN {X -0.114,Y -431.798,Z 859.673,A 0.000,B 0.000,C 90.000,E1 157.177} C_DIS
LIN {X 0.039,Y -441.207,Z 859.670,A 0.000,B 0.000,C 90.000,E1 156.538} C_DIS
LIN {X -0.093,Y -445.694,Z 859.668,A 0.000,B 0.000,C 90.000,E1 156.230} C_DIS
LIN {X -0.061,Y -450.334,Z 859.666,A 0.000,B 0.000,C 90.000,E1 155.869} C_DIS
LIN {X -0.006,Y -459.059,Z 859.662,A 0.000,B 0.000,C 90.000,E1 155.101} C_DIS
LIN {X -0.065,Y -463.460,Z 859.660,A 0.000,B 0.000,C 90.000,E1 154.717} C_DIS
LIN {X 0.120,Y -473.355,Z 859.654,A 0.000,B 0.000,C 90.000,E1 153.717} C_DIS
LIN {X 0.214,Y -478.643,Z 859.651,A 0.000,B 0.000,C 90.000,E1 153.127} C_DIS
LIN {X -0.112,Y -487.622,Z 859.645,A 0.000,B 0.000,C 90.000,E1 152.103} C_DIS
LIN {X -0.061,Y -500.583,Z 859.636,A 0.000,B 0.000,C 90.000,E1 150.461} C_DIS
LIN {X -0.158,Y -505.014,Z 859.633,A 0.000,B 0.000,C 90.000,E1 149.871} C_DIS
LIN {X 0.036,Y -509.264,Z 859.629,A 0.000,B 0.000,C 90.000,E1 149.253} C_DIS
LIN {X 0.053,Y -512.562,Z 859.627,A 0.000,B 0.000,C 90.000,E1 148.820} C_DIS
LIN {X 0.131,Y -517.316,Z 859.623,A 0.000,B 0.000,C 90.000,E1 148.074} C_DIS
LIN {X -0.116,Y -520.343,Z 859.620,A 0.000,B 0.000,C 90.000,E1 147.661} C_DIS
LIN {X 0.206,Y -523.852,Z 859.617,A 0.000,B 0.000,C 90.000,E1 147.041} C_DIS
LIN {X -0.007,Y -526.761,Z 859.615,A 0.000,B 0.000,C 90.000,E1 146.628} C_DIS
LIN {X 0.179,Y -534.178,Z 859.607,A 0.000,B 0.000,C 90.000,E1 145.308} C_DIS
LIN {X 0.023,Y -538.032,Z 859.603,A 0.000,B 0.000,C 90.000,E1 144.609} C_DIS
LIN {X -0.047,Y -544.791,Z 859.596,A 0.000,B 0.000,C 90.000,E1 143.336} C_DIS
LIN {X 0.126,Y -550.888,Z 859.590,A 0.000,B 0.000,C 90.000,E1 142.190} C_DIS
LIN {X -0.237,Y -561.525,Z 859.579,A 0.000,B 0.000,C 90.000,E1 140.275} C_DIS
LIN {X -0.143,Y -566.653,Z 859.574,A 0.000,B 0.000,C 90.000,E1 139.299} C_DIS
LIN {X -0.103,Y -570.175,Z 859.570,A 0.000,B 0.000,C 90.000,E1 138.609} C_DIS
LIN {X 0.067,Y -576.864,Z 859.563,A 0.000,B 0.000,C 90.000,E1 137.229} C_DIS
LIN {X -0.071,Y -583.543,Z 859.555,A 0.000,B 0.000,C 90.000,E1 135.891} C_DIS
LIN {X 0.269,Y -588.220,Z 859.550,A 0.000,B 0.000,C 90.000,E1 134.919} C_DIS
LIN {X 0.135,Y -593.279,Z 859.544,A 0.000,B 0.000,C 90.000,E1 133.866} C_DIS
LIN {X 0.062,Y -600.680,Z 859.535,A 0.000,B 0.000,C 90.000,E1 132.285} C_DIS
LIN {X -0.085,Y -606.409,Z 859.528,A 0.000,B 0.000,C 90.000,E1 130.987} C_DIS
LIN {X 0.050,Y -610.736,Z 859.522,A 0.000,B 0.000,C 90.000,E1 129.930} C_DIS
LIN {X 0.150,Y -615.808,Z 859.515,A 0.000,B 0.000,C 90.000,E1 128.624} C_DIS
LIN {X -0.284,Y -618.584,Z 859.510,A 0.000,B 0.000,C 90.000,E1 127.890} C_DIS
LIN {X -0.048,Y -623.123,Z 859.503,A 0.000,B 0.000,C 90.000,E1 126.583} C_DIS
LIN {X -0.086,Y -626.579,Z 859.498,A 0.000,B 0.000,C 90.000,E1 125.564} C_DIS
LIN {X -0.288,Y -628.986,Z 859.493,A 0.000,B 0.000,C 90.000,E1 124.818} C_DIS
LIN {X -0.103,Y -631.310,Z 859.489,A 0.000,B 0.000,C 90.000,E1 124.040} C_DIS
LIN {X 0.114,Y -633.812,Z 859.483,A 0.000,B 0.000,C 90.000,E1 123.007} C_DIS
LIN {X 0.024,Y -636.204,Z 859.478,A 0.000,B 0.000,C 90.000,E1 122.005} C_DIS
LIN {X -0.027,Y -638.247,Z 859.472,A 0.000,B 0.000,C 90.000,E1 121.003} C_DIS
LIN {X 0.004,Y -640.458,Z 859.465,A 0.000,B 0.000,C 90.000,E1 119.745} C_DIS
LIN {X 0.004,Y -642.023,Z 859.460,A 0.000,B 0.000,C 90.000,E1 118.743} C_DIS
LIN {X -0.291,Y -643.430,Z 859.454,A 0.000,B 0.000,C 90.000,E1 117.769} C_DIS
LIN {X -0.071,Y -644.379,Z 859.450,A 0.000,B 0.000,C 90.000,E1 117.001} C_DIS
LIN {X 0.159,Y -645.041,Z 859.446,A 0.000,B 0.000,C 90.000,E1 116.232} C_DIS
LIN {X -0.303,Y -645.773,Z 859.439,A 0.000,B 0.000,C 90.000,E1 115.027} C_DIS
LIN {X -0.064,Y -645.675,Z 859.435,A 0.000,B 0.000,C 90.000,E1 114.259} C_DIS
LIN {X 0.014,Y -645.616,Z 859.433,A 0.000,B 0.000,C 90.000,E1 114.003} C_DIS
LIN {X -0.169,Y -645.323,Z 859.432,A 0.000,B 0.000,C 90.000,E1 113.770} C_DIS
LIN {X -0.016,Y -644.016,Z 859.429,A 0.000,B 0.000,C 90.000,E1 113.259} C_DIS
LIN {X 0.242,Y -641.045,Z 859.426,A 0.000,B 0.000,C 90.000,E1 112.642} C_DIS
LIN {X 0.178,Y -636.793,Z 859.423,A 0.000,B 0.000,C 90.000,E1 112.153} C_DIS
LIN {X 0.212,Y -629.590,Z 859.420,A 0.000,B 0.000,C 90.000,E1 111.589} C_DIS
LIN {X -0.112,Y -622.773,Z 859.418,A 0.000,B 0.000,C 90.000,E1 111.227} C_DIS
LIN {X 0.052,Y -614.295,Z 859.416,A 0.000,B 0.000,C 90.000,E1 110.791} C_DIS
LIN {X -0.349,Y -599.041,Z 859.411,A 0.000,B 0.000,C 90.000,E1 110.066} C_DIS
LIN {X -0.030,Y -590.553,Z 859.409,A 0.000,B 0.000,C 90.000,E1 109.631} C_DIS
LIN {X 0.178,Y -583.535,Z 859.407,A 0.000,B 0.000,C 90.000,E1 109.322} C_DIS
LIN {X -0.107,Y -579.628,Z 859.407,A 0.000,B 0.000,C 90.000,E1 109.214} C_DIS
LIN {X 0.222,Y -572.314,Z 859.406,A 0.000,B 0.000,C 90.000,E1 108.960} C_DIS
LIN {X -0.150,Y -567.574,Z 859.405,A 0.000,B 0.000,C 90.000,E1 108.833} C_DIS
LIN {X -0.179,Y -566.195,Z 859.404,A 0.000,B 0.000,C 90.000,E1 108.779} C_DIS
LIN {X -0.300,Y -564.983,Z 859.404,A 0.000,B 0.000,C 90.000,E1 108.725} C_DIS
LIN {X 0.055,Y -562.836,Z 859.403,A 0.000,B 0.000,C 90.000,E1 108.489} C_DIS
LIN {X -0.163,Y -561.070,Z 859.401,A 0.000,B 0.000,C 90.000,E1 108.181} C_DIS
LIN {X -0.146,Y -560.107,Z 859.399,A 0.000,B 0.000,C 90.000,E1 107.764} C_DIS
LIN {X 0.147,Y -559.744,Z 859.397,A 0.000,B 0.000,C 90.000,E1 107.402} C_DIS
LIN {X -0.063,Y -559.520,Z 859.391,A 0.000,B 0.000,C 90.000,E1 106.315} C_DIS
LIN {X 0.170,Y -560.418,Z 859.374,A 0.000,B 0.000,C 90.000,E1 103.244} C_DIS
LIN {X -0.100,Y -561.938,Z 859.360,A 0.000,B 0.000,C 90.000,E1 100.782} C_DIS
LIN {X 0.194,Y -563.102,Z 859.351,A 0.000,B 0.000,C 90.000,E1 99.095} C_DIS
LIN {X -0.214,Y -564.079,Z 859.343,A 0.000,B 0.000,C 90.000,E1 97.757} C_DIS
LIN {X -0.131,Y -564.891,Z 859.335,A 0.000,B 0.000,C 90.000,E1 96.372} C_DIS
LIN {X -0.193,Y -565.420,Z 859.329,A 0.000,B 0.000,C 90.000,E1 95.277} C_DIS
LIN {X -0.146,Y -566.055,Z 859.322,A 0.000,B 0.000,C 90.000,E1 93.898} C_DIS
LIN {X -0.124,Y -566.526,Z 859.314,A 0.000,B 0.000,C 90.000,E1 92.522} C_DIS
LIN {X -0.091,Y -566.887,Z 859.306,A 0.000,B 0.000,C 90.000,E1 91.146} C_DIS
LIN {X -0.065,Y -567.252,Z 859.299,A 0.000,B 0.000,C 90.000,E1 89.771} C_DIS
LIN {X 0.102,Y -567.622,Z 859.290,A 0.000,B 0.000,C 90.000,E1 88.108} C_DIS
LIN {X 0.279,Y -567.908,Z 859.280,A 0.000,B 0.000,C 90.000,E1 86.445} C_DIS
LIN {X -0.080,Y -568.173,Z 859.271,A 0.000,B 0.000,C 90.000,E1 84.837} C_DIS
LIN {X 0.182,Y -568.471,Z 859.262,A 0.000,B 0.000,C 90.000,E1 83.166} C_DIS
LIN {X 0.229,Y -569.055,Z 859.250,A 0.000,B 0.000,C 90.000,E1 80.971} C_DIS
LIN {X -0.273,Y -569.729,Z 859.239,A 0.000,B 0.000,C 90.000,E1 79.106} C_DIS
LIN {X -0.083,Y -570.493,Z 859.229,A 0.000,B 0.000,C 90.000,E1 77.173} C_DIS
LIN {X -0.121,Y -570.995,Z 859.221,A 0.000,B 0.000,C 90.000,E1 75.811} C_DIS
LIN {X -0.146,Y -571.347,Z 859.214,A 0.000,B 0.000,C 90.000,E1 74.448} C_DIS
LIN {X -0.174,Y -571.627,Z 859.206,A 0.000,B 0.000,C 90.000,E1 73.087} C_DIS
LIN {X -0.238,Y -571.827,Z 859.197,A 0.000,B 0.000,C 90.000,E1 71.456} C_DIS
LIN {X -0.123,Y -571.833,Z 859.185,A 0.000,B 0.000,C 90.000,E1 69.263} C_DIS
LIN {X 0.005,Y -571.791,Z 859.176,A 0.000,B 0.000,C 90.000,E1 67.614} C_DIS
LIN {X 0.042,Y -571.668,Z 859.167,A 0.000,B 0.000,C 90.000,E1 65.973} C_DIS
LIN {X 0.252,Y -571.444,Z 859.159,A 0.000,B 0.000,C 90.000,E1 64.588} C_DIS
LIN {X -0.231,Y -570.993,Z 859.150,A 0.000,B 0.000,C 90.000,E1 62.999} C_DIS
LIN {X -0.300,Y -570.532,Z 859.142,A 0.000,B 0.000,C 90.000,E1 61.641} C_DIS
LIN {X -0.211,Y -570.006,Z 859.136,A 0.000,B 0.000,C 90.000,E1 60.539} C_DIS
LIN {X 0.326,Y -569.594,Z 859.132,A 0.000,B 0.000,C 90.000,E1 59.665} C_DIS
LIN {X 0.012,Y -568.487,Z 859.124,A 0.000,B 0.000,C 90.000,E1 58.329} C_DIS
LIN {X 0.058,Y -567.808,Z 859.120,A 0.000,B 0.000,C 90.000,E1 57.502} C_DIS
LIN {X -0.211,Y -566.925,Z 859.115,A 0.000,B 0.000,C 90.000,E1 56.707} C_DIS
LIN {X -0.071,Y -565.516,Z 859.109,A 0.000,B 0.000,C 90.000,E1 55.595} C_DIS
LIN {X -0.058,Y -564.371,Z 859.104,A 0.000,B 0.000,C 90.000,E1 54.769} C_DIS
LIN {X 0.039,Y -562.677,Z 859.098,A 0.000,B 0.000,C 90.000,E1 53.657} C_DIS
LIN {X -0.006,Y -560.668,Z 859.092,A 0.000,B 0.000,C 90.000,E1 52.557} C_DIS
LIN {X -0.162,Y -558.987,Z 859.087,A 0.000,B 0.000,C 90.000,E1 51.743} C_DIS
LIN {X 0.018,Y -557.782,Z 859.084,A 0.000,B 0.000,C 90.000,E1 51.170} C_DIS
LIN {X -0.167,Y -555.686,Z 859.080,A 0.000,B 0.000,C 90.000,E1 50.356} C_DIS
LIN {X 0.053,Y -552.320,Z 859.073,A 0.000,B 0.000,C 90.000,E1 49.218} C_DIS
LIN {X -0.244,Y -550.473,Z 859.070,A 0.000,B 0.000,C 90.000,E1 48.690} C_DIS
LIN {X 0.222,Y -548.440,Z 859.067,A 0.000,B 0.000,C 90.000,E1 48.081} C_DIS
LIN {X 0.298,Y -545.087,Z 859.063,A 0.000,B 0.000,C 90.000,E1 47.229} C_DIS
LIN {X 0.142,Y -542.034,Z 859.059,A 0.000,B 0.000,C 90.000,E1 46.539} C_DIS
LIN {X -0.248,Y -538.003,Z 859.054,A 0.000,B 0.000,C 90.000,E1 45.729} C_DIS
LIN {X 0.302,Y -535.796,Z 859.052,A 0.000,B 0.000,C 90.000,E1 45.243} C_DIS
LIN {X 0.255,Y -532.584,Z 859.048,A 0.000,B 0.000,C 90.000,E1 44.676} C_DIS
LIN {X 0.186,Y -529.098,Z 859.045,A 0.000,B 0.000,C 90.000,E1 44.109} C_DIS
LIN {X 0.091,Y -525.316,Z 859.042,A 0.000,B 0.000,C 90.000,E1 43.542} C_DIS
LIN {X -0.033,Y -521.319,Z 859.039,A 0.000,B 0.000,C 90.000,E1 42.975} C_DIS
LIN {X 0.059,Y -518.162,Z 859.036,A 0.000,B 0.000,C 90.000,E1 42.528} C_DIS
LIN {X -0.248,Y -512.461,Z 859.032,A 0.000,B 0.000,C 90.000,E1 41.838} C_DIS
LIN {X -0.159,Y -508.897,Z 859.030,A 0.000,B 0.000,C 90.000,E1 41.391} C_DIS
LIN {X -0.059,Y -505.155,Z 859.027,A 0.000,B 0.000,C 90.000,E1 40.943} C_DIS
LIN {X -0.079,Y -498.447,Z 859.023,A 0.000,B 0.000,C 90.000,E1 40.216} C_DIS
LIN {X 0.087,Y -494.250,Z 859.021,A 0.000,B 0.000,C 90.000,E1 39.769} C_DIS
LIN {X 0.256,Y -488.524,Z 859.018,A 0.000,B 0.000,C 90.000,E1 39.197} C_DIS
LIN {X 0.119,Y -481.257,Z 859.014,A 0.000,B 0.000,C 90.000,E1 38.543} C_DIS
LIN {X -0.064,Y -470.797,Z 859.009,A 0.000,B 0.000,C 90.000,E1 37.684} C_DIS
LIN {X -0.196,Y -463.049,Z 859.006,A 0.000,B 0.000,C 90.000,E1 37.076} C_DIS
LIN {X -0.110,Y -450.521,Z 859.000,A 0.000,B 0.000,C 90.000,E1 36.091} C_DIS
LIN {X 0.037,Y -436.395,Z 858.994,A 0.000,B 0.000,C 90.000,E1 34.978} C_DIS
LIN {X 0.134,Y -417.960,Z 858.986,A 0.000,B 0.000,C 90.000,E1 33.452} C_DIS
LIN {X 0.088,Y -404.373,Z 858.979,A 0.000,B 0.000,C 90.000,E1 32.212} C_DIS
LIN {X -0.125,Y -400.092,Z 858.977,A 0.000,B 0.000,C 90.000,E1 31.799} C_DIS
LIN {X -0.170,Y -397.873,Z 858.975,A 0.000,B 0.000,C 90.000,E1 31.544} C_DIS
LIN {X 0.037,Y -394.798,Z 858.973,A 0.000,B 0.000,C 90.000,E1 31.082} C_DIS
LIN {X -0.090,Y -393.744,Z 858.972,A 0.000,B 0.000,C 90.000,E1 30.924} C_DIS
LIN {X 0.107,Y -391.705,Z 858.969,A 0.000,B 0.000,C 90.000,E1 30.463} C_DIS
LIN {X -0.107,Y -390.626,Z 858.967,A 0.000,B 0.000,C 90.000,E1 30.050} C_DIS
LIN {X -0.065,Y -389.959,Z 858.962,A 0.000,B 0.000,C 90.000,E1 29.155} C_DIS
LIN {X -0.027,Y -389.813,Z 858.958,A 0.000,B 0.000,C 90.000,E1 28.437} C_DIS
LIN {X 0.141,Y -391.723,Z 858.940,A 0.000,B 0.000,C 90.000,E1 25.207} C_DIS
LIN {X 0.133,Y -393.402,Z 858.928,A 0.000,B 0.000,C 90.000,E1 23.078} C_DIS
LIN {X 0.072,Y -395.694,Z 858.915,A 0.000,B 0.000,C 90.000,E1 20.610} C_DIS
LIN {X -0.050,Y -399.065,Z 858.897,A 0.000,B 0.000,C 90.000,E1 17.457} C_DIS
LIN {X -0.022,Y -402.964,Z 858.879,A 0.000,B 0.000,C 90.000,E1 14.300} C_DIS
LIN {X -0.161,Y -406.436,Z 858.866,A 0.000,B 0.000,C 90.000,E1 11.883} C_DIS
LIN {X -0.091,Y -409.135,Z 858.856,A 0.000,B 0.000,C 90.000,E1 10.141} C_DIS
LIN {X 0.077,Y -412.536,Z 858.845,A 0.000,B 0.000,C 90.000,E1 8.049} C_DIS
LIN {X -0.150,Y -416.777,Z 858.831,A 0.000,B 0.000,C 90.000,E1 5.682} C_DIS
LIN {X 0.171,Y -422.618,Z 858.815,A 0.000,B 0.000,C 90.000,E1 2.579} C_DIS
LIN {X -0.199,Y -429.601,Z 858.797,A 0.000,B 0.000,C 90.000,E1 359.484} C_DIS
LIN {X 0.041,Y -436.032,Z 858.782,A 0.000,B 0.000,C 90.000,E1 356.788} C_DIS
LIN {X 0.079,Y -442.996,Z 858.768,A 0.000,B 0.000,C 90.000,E1 354.147} C_DIS
LIN {X -0.092,Y -445.309,Z 858.764,A 0.000,B 0.000,C 90.000,E1 353.514} C_DIS
LIN {X -0.048,Y -447.205,Z 858.762,A 0.000,B 0.000,C 90.000,E1 353.109} C_DIS
LIN {X 0.193,Y -451.037,Z 858.759,A 0.000,B 0.000,C 90.000,E1 352.591} C_DIS
LIN {X 0.118,Y -452.422,Z 858.758,A 0.000,B 0.000,C 90.000,E1 352.470} C_DIS
LIN {X -0.034,Y -455.879,Z 858.757,A 0.000,B 0.000,C 90.000,E1 352.243} C_DIS
LIN {X -0.053,Y -457.759,Z 858.756,A 0.000,B 0.000,C 90.000,E1 352.129} C_DIS
LIN {X -0.139,Y -477.044,Z 858.751,A 0.000,B 0.000,C 90.000,E1 351.197} C_DIS
LIN {X -0.107,Y -483.370,Z 858.749,A 0.000,B 0.000,C 90.000,E1 350.849} C_DIS
LIN {X -0.231,Y -491.488,Z 858.747,A 0.000,B 0.000,C 90.000,E1 350.387} C_DIS
LIN {X 0.150,Y -499.462,Z 858.744,A 0.000,B 0.000,C 90.000,E1 349.859} C_DIS
LIN {X -0.071,Y -512.175,Z 858.739,A 0.000,B 0.000,C 90.000,E1 349.050} C_DIS
LIN {X -0.049,Y -521.387,Z 858.736,A 0.000,B 0.000,C 90.000,E1 348.409} C_DIS
LIN {X -0.184,Y -530.515,Z 858.732,A 0.000,B 0.000,C 90.000,E1 347.757} C_DIS
LIN {X -0.139,Y -540.707,Z 858.727,A 0.000,B 0.000,C 90.000,E1 346.937} C_DIS
LIN {X 0.167,Y -549.176,Z 858.723,A 0.000,B 0.000,C 90.000,E1 346.172} C_DIS
LIN {X -0.129,Y -554.495,Z 858.721,A 0.000,B 0.000,C 90.000,E1 345.700} C_DIS
LIN {X -0.020,Y -560.983,Z 858.717,A 0.000,B 0.000,C 90.000,E1 345.046} C_DIS
LIN {X -0.081,Y -565.995,Z 858.714,A 0.000,B 0.000,C 90.000,E1 344.519} C_DIS
LIN {X 0.304,Y -572.091,Z 858.710,A 0.000,B 0.000,C 90.000,E1 343.795} C_DIS
LIN {X 0.122,Y -576.557,Z 858.707,A 0.000,B 0.000,C 90.000,E1 343.268} C_DIS
LIN {X -0.297,Y -583.918,Z 858.702,A 0.000,B 0.000,C 90.000,E1 342.362} C_DIS
LIN {X -0.233,Y -587.817,Z 858.699,A 0.000,B 0.000,C 90.000,E1 341.819} C_DIS
LIN {X -0.140,Y -591.446,Z 858.696,A 0.000,B 0.000,C 90.000,E1 341.275} C_DIS
LIN {X 0.175,Y -597.391,Z 858.691,A 0.000,B 0.000,C 90.000,E1 340.315} C_DIS
LIN {X 0.200,Y -602.882,Z 858.686,A 0.000,B 0.000,C 90.000,E1 339.390} C_DIS
LIN {X 0.017,Y -609.534,Z 858.679,A 0.000,B 0.000,C 90.000,E1 338.230} C_DIS
LIN {X -0.357,Y -613.798,Z 858.675,A 0.000,B 0.000,C 90.000,E1 337.486} C_DIS
LIN {X 0.102,Y -619.172,Z 858.669,A 0.000,B 0.000,C 90.000,E1 336.410} C_DIS
LIN {X -0.176,Y -623.593,Z 858.664,A 0.000,B 0.000,C 90.000,E1 335.537} C_DIS
LIN {X 0.172,Y -629.419,Z 858.657,A 0.000,B 0.000,C 90.000,E1 334.229} C_DIS
LIN {X 0.218,Y -631.599,Z 858.654,A 0.000,B 0.000,C 90.000,E1 333.717} C_DIS
LIN {X -0.209,Y -635.709,Z 858.648,A 0.000,B 0.000,C 90.000,E1 332.743} C_DIS
LIN {X -0.017,Y -639.625,Z 858.643,A 0.000,B 0.000,C 90.000,E1 331.719} C_DIS
LIN {X 0.037,Y -644.154,Z 858.636,A 0.000,B 0.000,C 90.000,E1 330.461} C_DIS
LIN {X 0.094,Y -647.627,Z 858.630,A 0.000,B 0.000,C 90.000,E1 329.459} C_DIS
LIN {X 0.199,Y -650.806,Z 858.625,A 0.000,B 0.000,C 90.000,E1 328.456} C_DIS
LIN {X 0.345,Y -653.768,Z 858.619,A 0.000,B 0.000,C 90.000,E1 327.454} C_DIS
LIN {X 0.430,Y -657.177,Z 858.613,A 0.000,B 0.000,C 90.000,E1 326.215} C_DIS
LIN {X 0.028,Y -660.176,Z 858.606,A 0.000,B 0.000,C 90.000,E1 325.022} C_DIS
LIN {X 0.164,Y -661.817,Z 858.602,A 0.000,B 0.000,C 90.000,E1 324.276} C_DIS
LIN {X -0.272,Y -663.784,Z 858.596,A 0.000,B 0.000,C 90.000,E1 323.336} C_DIS
LIN {X -0.153,Y -665.533,Z 858.591,A 0.000,B 0.000,C 90.000,E1 322.351} C_DIS
LIN {X -0.057,Y -667.749,Z 858.583,A 0.000,B 0.000,C 90.000,E1 320.884} C_DIS
LIN {X 0.001,Y -669.013,Z 858.577,A 0.000,B 0.000,C 90.000,E1 319.908} C_DIS
LIN {X 0.089,Y -670.693,Z 858.569,A 0.000,B 0.000,C 90.000,E1 318.447} C_DIS
LIN {X -0.210,Y -673.018,Z 858.559,A 0.000,B 0.000,C 90.000,E1 316.539} C_DIS
LIN {X -0.098,Y -674.561,Z 858.552,A 0.000,B 0.000,C 90.000,E1 315.324} C_DIS
LIN {X -0.045,Y -674.939,Z 858.549,A 0.000,B 0.000,C 90.000,E1 314.838} C_DIS
LIN {X -0.017,Y -675.250,Z 858.548,A 0.000,B 0.000,C 90.000,E1 314.595} C_DIS
LIN {X -0.241,Y -677.098,Z 858.537,A 0.000,B 0.000,C 90.000,E1 312.690} C_DIS
LIN {X -0.029,Y -678.290,Z 858.530,A 0.000,B 0.000,C 90.000,E1 311.472} C_DIS
LIN {X 0.239,Y -679.637,Z 858.522,A 0.000,B 0.000,C 90.000,E1 310.011} C_DIS
LIN {X 0.052,Y -680.678,Z 858.516,A 0.000,B 0.000,C 90.000,E1 308.830} C_DIS
LIN {X 0.055,Y -682.077,Z 858.506,A 0.000,B 0.000,C 90.000,E1 307.156} C_DIS
LIN {X 0.056,Y -683.205,Z 858.499,A 0.000,B 0.000,C 90.000,E1 305.724} C_DIS
LIN {X -0.324,Y -684.174,Z 858.491,A 0.000,B 0.000,C 90.000,E1 304.326} C_DIS
LIN {X 0.256,Y -684.972,Z 858.484,A 0.000,B 0.000,C 90.000,E1 303.086} C_DIS
LIN {X -0.057,Y -686.367,Z 858.473,A 0.000,B 0.000,C 90.000,E1 301.209} C_DIS
LIN {X -0.112,Y -688.085,Z 858.462,A 0.000,B 0.000,C 90.000,E1 299.077} C_DIS
LIN {X 0.048,Y -689.393,Z 858.454,A 0.000,B 0.000,C 90.000,E1 297.641} C_DIS
LIN {X 0.391,Y -691.277,Z 858.443,A 0.000,B 0.000,C 90.000,E1 295.720} C_DIS
LIN {X -0.246,Y -692.418,Z 858.437,A 0.000,B 0.000,C 90.000,E1 294.591} C_DIS
LIN {X -0.153,Y -692.887,Z 858.433,A 0.000,B 0.000,C 90.000,E1 293.875} C_DIS
LIN {X 0.050,Y -692.856,Z 858.430,A 0.000,B 0.000,C 90.000,E1 293.387} C_DIS
LIN {X 0.019,Y -692.644,Z 858.429,A 0.000,B 0.000,C 90.000,E1 293.153} C_DIS
LIN {X 0.259,Y -692.142,Z 858.427,A 0.000,B 0.000,C 90.000,E1 292.898} C_DIS
LIN {X -0.140,Y -691.499,Z 858.426,A 0.000,B 0.000,C 90.000,E1 292.695} C_DIS
LIN {X -0.171,Y -690.513,Z 858.425,A 0.000,B 0.000,C 90.000,E1 292.461} C_DIS
LIN {X 0.173,Y -687.758,Z 858.423,A 0.000,B 0.000,C 90.000,E1 292.078} C_DIS
LIN {X 0.137,Y -685.540,Z 858.421,A 0.000,B 0.000,C 90.000,E1 291.844} C_DIS
LIN {X 0.244,Y -683.907,Z 858.421,A 0.000,B 0.000,C 90.000,E1 291.716} C_DIS
LIN {X -0.011,Y -679.507,Z 858.420,A 0.000,B 0.000,C 90.000,E1 291.535} C_DIS
LIN {X -0.138,Y -674.007,Z 858.419,A 0.000,B 0.000,C 90.000,E1 291.334} C_DIS
LIN {X -0.329,Y -670.102,Z 858.418,A 0.000,B 0.000,C 90.000,E1 291.227} C_DIS
LIN {X -0.009,Y -655.400,Z 858.416,A 0.000,B 0.000,C 90.000,E1 290.865} C_DIS
LIN {X 0.309,Y -649.177,Z 858.415,A 0.000,B 0.000,C 90.000,E1 290.610} C_DIS
LIN {X 0.215,Y -647.744,Z 858.414,A 0.000,B 0.000,C 90.000,E1 290.556} C_DIS
LIN {X -0.300,Y -644.650,Z 858.413,A 0.000,B 0.000,C 90.000,E1 290.429} C_DIS
LIN {X -0.361,Y -644.594,Z 858.413,A 0.000,B 0.000,C 90.000,E1 290.429} C_DIS
LIN {X 0.104,Y -643.081,Z 858.412,A 0.000,B 0.000,C 90.000,E1 290.194} C_DIS
LIN {X 0.060,Y -643.076,Z 858.412,A 0.000,B 0.000,C 90.000,E1 290.194} C_DIS
LIN {X 0.177,Y -643.075,Z 858.412,A 0.000,B 0.000,C 90.000,E1 290.066} C_DIS
LIN {X 0.205,Y -643.365,Z 858.411,A 0.000,B 0.000,C 90.000,E1 289.939} C_DIS
LIN {X 0.094,Y -645.418,Z 858.408,A 0.000,B 0.000,C 90.000,E1 289.450} C_DIS
LIN {X -0.230,Y -652.114,Z 858.401,A 0.000,B 0.000,C 90.000,E1 288.236} C_DIS
LIN {X 0.044,Y -656.237,Z 858.396,A 0.000,B 0.000,C 90.000,E1 287.347} C_DIS
LIN {X 0.004,Y -658.387,Z 858.394,A 0.000,B 0.000,C 90.000,E1 286.858} C_DIS
LIN {X -0.132,Y -661.199,Z 858.390,A 0.000,B 0.000,C 90.000,E1 286.134} C_DIS
LIN {X 0.307,Y -662.793,Z 858.387,A 0.000,B 0.000,C 90.000,E1 285.607} C_DIS
LIN {X 0.035,Y -664.791,Z 858.383,A 0.000,B 0.000,C 90.000,E1 284.898} C_DIS
LIN {X 0.031,Y -665.893,Z 858.380,A 0.000,B 0.000,C 90.000,E1 284.411} C_DIS
LIN {X -0.217,Y -667.117,Z 858.376,A 0.000,B 0.000,C 90.000,E1 283.703} C_DIS
LIN {X 0.274,Y -667.746,Z 858.373,A 0.000,B 0.000,C 90.000,E1 283.175} C_DIS
LIN {X -0.102,Y -668.347,Z 858.369,A 0.000,B 0.000,C 90.000,E1 282.479} C_DIS
LIN {X -0.251,Y -668.613,Z 858.367,A 0.000,B 0.000,C 90.000,E1 282.007} C_DIS
LIN {X 0.255,Y -668.668,Z 858.364,A 0.000,B 0.000,C 90.000,E1 281.478} C_DIS
LIN {X -0.101,Y -668.242,Z 858.360,A 0.000,B 0.000,C 90.000,E1 280.782} C_DIS
LIN {X -0.257,Y -667.739,Z 858.357,A 0.000,B 0.000,C 90.000,E1 280.310} C_DIS
LIN {X 0.122,Y -666.978,Z 858.354,A 0.000,B 0.000,C 90.000,E1 279.792} C_DIS
LIN {X -0.048,Y -665.919,Z 858.352,A 0.000,B 0.000,C 90.000,E1 279.321} C_DIS
LIN {X -0.334,Y -664.568,Z 858.349,A 0.000,B 0.000,C 90.000,E1 278.859} C_DIS
LIN {X 0.032,Y -662.848,Z 858.346,A 0.000,B 0.000,C 90.000,E1 278.341} C_DIS
LIN {X -0.175,Y -660.770,Z 858.344,A 0.000,B 0.000,C 90.000,E1 277.871} C_DIS
LIN {X 0.281,Y -659.705,Z 858.342,A 0.000,B 0.000,C 90.000,E1 277.587} C_DIS
LIN {X -0.036,Y -657.170,Z 858.340,A 0.000,B 0.000,C 90.000,E1 277.125} C_DIS
LIN {X 0.247,Y -653.472,Z 858.336,A 0.000,B 0.000,C 90.000,E1 276.486} C_DIS
LIN {X -0.184,Y -650.082,Z 858.333,A 0.000,B 0.000,C 90.000,E1 276.030} C_DIS
LIN {X 0.031,Y -644.978,Z 858.330,A 0.000,B 0.000,C 90.000,E1 275.391} C_DIS
LIN {X 0.254,Y -640.237,Z 858.327,A 0.000,B 0.000,C 90.000,E1 274.878} C_DIS
LIN {X 0.000,Y -634.840,Z 858.325,A 0.000,B 0.000,C 90.000,E1 274.416} C_DIS
LIN {X -0.296,Y -631.028,Z 858.323,A 0.000,B 0.000,C 90.000,E1 274.131} C_DIS
LIN {X 0.075,Y -625.194,Z 858.320,A 0.000,B 0.000,C 90.000,E1 273.669} C_DIS
LIN {X 0.261,Y -617.480,Z 858.318,A 0.000,B 0.000,C 90.000,E1 273.154} C_DIS
LIN {X -0.055,Y -610.974,Z 858.316,A 0.000,B 0.000,C 90.000,E1 272.808} C_DIS
LIN {X -0.263,Y -602.210,Z 858.313,A 0.000,B 0.000,C 90.000,E1 272.407} C_DIS
LIN {X -0.248,Y -596.980,Z 858.312,A 0.000,B 0.000,C 90.000,E1 272.178} C_DIS
LIN {X 0.010,Y -591.285,Z 858.311,A 0.000,B 0.000,C 90.000,E1 271.949} C_DIS
LIN {X 0.087,Y -583.838,Z 858.310,A 0.000,B 0.000,C 90.000,E1 271.718} C_DIS
LIN {X -0.113,Y -578.035,Z 858.309,A 0.000,B 0.000,C 90.000,E1 271.604} C_DIS
LIN {X -0.081,Y -570.926,Z 858.308,A 0.000,B 0.000,C 90.000,E1 271.489} C_DIS
LIN {X -0.078,Y -564.150,Z 858.308,A 0.000,B 0.000,C 90.000,E1 271.432} C_DIS
LIN {X 0.138,Y -555.472,Z 858.308,A 0.000,B 0.000,C 90.000,E1 271.375} C_DIS
LIN {X -0.008,Y -552.954,Z 858.308,A 0.000,B 0.000,C 90.000,E1 271.375} C_DIS
LIN {X 0.082,Y -549.452,Z 858.307,A 0.000,B 0.000,C 90.000,E1 271.260} C_DIS
LIN {X 0.048,Y -549.372,Z 858.307,A 0.000,B 0.000,C 90.000,E1 271.260} C_DIS
LIN {X -0.062,Y -548.482,Z 858.306,A 0.000,B 0.000,C 90.000,E1 271.088} C_DIS
LIN {X -0.056,Y -547.394,Z 858.305,A 0.000,B 0.000,C 90.000,E1 270.917} C_DIS
LIN {X -0.098,Y -547.366,Z 858.305,A 0.000,B 0.000,C 90.000,E1 270.917} C_DIS
LIN {X -0.214,Y -546.461,Z 858.302,A 0.000,B 0.000,C 90.000,E1 270.401} C_DIS
LIN {X 0.223,Y -543.728,Z 858.285,A 0.000,B 0.000,C 90.000,E1 267.249} C_DIS
LIN {X -0.092,Y -542.601,Z 858.275,A 0.000,B 0.000,C 90.000,E1 265.584} C_DIS
LIN {X 0.159,Y -541.406,Z 858.266,A 0.000,B 0.000,C 90.000,E1 263.856} C_DIS
LIN {X 0.241,Y -540.697,Z 858.261,A 0.000,B 0.000,C 90.000,E1 262.996} C_DIS
LIN {X -0.022,Y -539.383,Z 858.253,A 0.000,B 0.000,C 90.000,E1 261.602} C_DIS
LIN {X 0.234,Y -538.136,Z 858.245,A 0.000,B 0.000,C 90.000,E1 260.151} C_DIS
LIN {X -0.069,Y -536.733,Z 858.238,A 0.000,B 0.000,C 90.000,E1 258.757} C_DIS
LIN {X -0.298,Y -535.227,Z 858.230,A 0.000,B 0.000,C 90.000,E1 257.353} C_DIS
LIN {X 0.036,Y -533.872,Z 858.223,A 0.000,B 0.000,C 90.000,E1 256.172} C_DIS
LIN {X 0.091,Y -531.404,Z 858.212,A 0.000,B 0.000,C 90.000,E1 254.157} C_DIS
LIN {X 0.205,Y -529.403,Z 858.203,A 0.000,B 0.000,C 90.000,E1 252.417} C_DIS
LIN {X 0.089,Y -527.982,Z 858.196,A 0.000,B 0.000,C 90.000,E1 251.275} C_DIS
LIN {X 0.115,Y -526.062,Z 858.188,A 0.000,B 0.000,C 90.000,E1 249.826} C_DIS
LIN {X -0.209,Y -524.156,Z 858.180,A 0.000,B 0.000,C 90.000,E1 248.411} C_DIS
LIN {X -0.206,Y -521.551,Z 858.170,A 0.000,B 0.000,C 90.000,E1 246.666} C_DIS
LIN {X -0.077,Y -519.773,Z 858.164,A 0.000,B 0.000,C 90.000,E1 245.485} C_DIS
LIN {X -0.096,Y -517.507,Z 858.156,A 0.000,B 0.000,C 90.000,E1 244.024} C_DIS
LIN {X 0.057,Y -516.020,Z 858.151,A 0.000,B 0.000,C 90.000,E1 243.127} C_DIS
LIN {X -0.147,Y -512.921,Z 858.141,A 0.000,B 0.000,C 90.000,E1 241.385} C_DIS
LIN {X -0.160,Y -510.924,Z 858.134,A 0.000,B 0.000,C 90.000,E1 240.205} C_DIS
LIN {X 0.017,Y -507.557,Z 858.125,A 0.000,B 0.000,C 90.000,E1 238.408} C_DIS
LIN {X 0.067,Y -504.658,Z 858.116,A 0.000,B 0.000,C 90.000,E1 236.914} C_DIS
LIN {X 0.153,Y -502.819,Z 858.111,A 0.000,B 0.000,C 90.000,E1 236.008} C_DIS
LIN {X 0.221,Y -500.896,Z 858.106,A 0.000,B 0.000,C 90.000,E1 235.102} C_DIS
LIN {X 0.143,Y -498.078,Z 858.100,A 0.000,B 0.000,C 90.000,E1 233.909} C_DIS
LIN {X -0.102,Y -493.079,Z 858.088,A 0.000,B 0.000,C 90.000,E1 231.823} C_DIS
LIN {X 0.137,Y -488.082,Z 858.076,A 0.000,B 0.000,C 90.000,E1 229.666} C_DIS
LIN {X -0.086,Y -484.601,Z 858.068,A 0.000,B 0.000,C 90.000,E1 228.162} C_DIS
LIN {X 0.199,Y -479.868,Z 858.056,A 0.000,B 0.000,C 90.000,E1 225.972} C_DIS
LIN {X 0.012,Y -475.226,Z 858.044,A 0.000,B 0.000,C 90.000,E1 223.824} C_DIS
LIN {X -0.068,Y -471.146,Z 858.033,A 0.000,B 0.000,C 90.000,E1 221.962} C_DIS
LIN {X -0.177,Y -467.099,Z 858.023,A 0.000,B 0.000,C 90.000,E1 220.092} C_DIS
LIN {X -0.012,Y -463.132,Z 858.012,A 0.000,B 0.000,C 90.000,E1 218.177} C_DIS
LIN {X -0.226,Y -459.185,Z 858.002,A 0.000,B 0.000,C 90.000,E1 216.297} C_DIS
LIN {X 0.025,Y -453.631,Z 857.987,A 0.000,B 0.000,C 90.000,E1 213.706} C_DIS
LIN {X -0.105,Y -448.837,Z 857.975,A 0.000,B 0.000,C 90.000,E1 211.465} C_DIS
LIN {X -0.155,Y -443.338,Z 857.960,A 0.000,B 0.000,C 90.000,E1 208.871} C_DIS
LIN {X 0.106,Y -439.286,Z 857.949,A 0.000,B 0.000,C 90.000,E1 206.873} C_DIS
LIN {X 0.076,Y -435.176,Z 857.938,A 0.000,B 0.000,C 90.000,E1 204.899} C_DIS
LIN {X 0.164,Y -431.104,Z 857.927,A 0.000,B 0.000,C 90.000,E1 202.898} C_DIS
LIN {X 0.183,Y -427.766,Z 857.918,A 0.000,B 0.000,C 90.000,E1 201.227} C_DIS
LIN {X -0.016,Y -424.476,Z 857.909,A 0.000,B 0.000,C 90.000,E1 199.577} C_DIS
LIN {X -0.236,Y -420.543,Z 857.898,A 0.000,B 0.000,C 90.000,E1 197.583} C_DIS
LIN {X -0.076,Y -417.970,Z 857.890,A 0.000,B 0.000,C 90.000,E1 196.205} C_DIS
LIN {X 0.033,Y -415.133,Z 857.882,A 0.000,B 0.000,C 90.000,E1 194.828} C_DIS
LIN {X 0.017,Y -411.589,Z 857.873,A 0.000,B 0.000,C 90.000,E1 193.119} C_DIS
LIN {X -0.036,Y -406.973,Z 857.860,A 0.000,B 0.000,C 90.000,E1 190.715} C_DIS
LIN {X 0.021,Y -403.600,Z 857.850,A 0.000,B 0.000,C 90.000,E1 188.973} C_DIS
LIN {X -0.077,Y -398.783,Z 857.836,A 0.000,B 0.000,C 90.000,E1 186.543} C_DIS
LIN {X 0.188,Y -392.681,Z 857.817,A 0.000,B 0.000,C 90.000,E1 182.980} C_DIS
LIN {X -0.060,Y -388.607,Z 857.801,A 0.000,B 0.000,C 90.000,E1 180.172} C_DIS
LIN {X -0.137,Y -386.141,Z 857.791,A 0.000,B 0.000,C 90.000,E1 178.396} C_DIS
LIN {X 0.030,Y -383.100,Z 857.779,A 0.000,B 0.000,C 90.000,E1 176.216} C_DIS
LIN {X -0.009,Y -381.099,Z 857.771,A 0.000,B 0.000,C 90.000,E1 174.780} C_DIS
LIN {X -0.105,Y -377.377,Z 857.755,A 0.000,B 0.000,C 90.000,E1 171.894} C_DIS
LIN {X 0.084,Y -373.106,Z 857.729,A 0.000,B 0.000,C 90.000,E1 167.117} C_DIS
LIN {X 0.120,Y -372.375,Z 857.720,A 0.000,B 0.000,C 90.000,E1 165.644} C_DIS
LIN {X -0.049,Y -372.377,Z 857.716,A 0.000,B 0.000,C 90.000,E1 164.936} C_DIS
LIN {X -0.119,Y -372.334,Z 857.712,A 0.000,B 0.000,C 90.000,E1 164.212} C_DIS
LIN {X 0.068,Y -372.501,Z 857.708,A 0.000,B 0.000,C 90.000,E1 163.449} C_DIS
LIN {X 0.002,Y -372.890,Z 857.704,A 0.000,B 0.000,C 90.000,E1 162.725} C_DIS
LIN {X 0.042,Y -373.802,Z 857.700,A 0.000,B 0.000,C 90.000,E1 162.000} C_DIS
LIN {X 0.133,Y -374.323,Z 857.699,A 0.000,B 0.000,C 90.000,E1 161.764} C_DIS
LIN {X 0.083,Y -375.657,Z 857.695,A 0.000,B 0.000,C 90.000,E1 161.040} C_DIS
LIN {X 0.072,Y -376.097,Z 857.694,A 0.000,B 0.000,C 90.000,E1 160.859} C_DIS
LIN {X -0.100,Y -377.573,Z 857.692,A 0.000,B 0.000,C 90.000,E1 160.477} C_DIS
LIN {X -0.108,Y -378.131,Z 857.690,A 0.000,B 0.000,C 90.000,E1 160.296} C_DIS
LIN {X -0.114,Y -378.862,Z 857.689,A 0.000,B 0.000,C 90.000,E1 160.115} C_DIS
LIN {X -0.099,Y -382.028,Z 857.686,A 0.000,B 0.000,C 90.000,E1 159.518} C_DIS
LIN {X -0.098,Y -383.243,Z 857.685,A 0.000,B 0.000,C 90.000,E1 159.337} C_DIS
LIN {X -0.080,Y -387.557,Z 857.683,A 0.000,B 0.000,C 90.000,E1 158.901} C_DIS
LIN {X 0.143,Y -389.211,Z 857.682,A 0.000,B 0.000,C 90.000,E1 158.720} C_DIS
LIN {X -0.066,Y -395.105,Z 857.680,A 0.000,B 0.000,C 90.000,E1 158.411} C_DIS
LIN {X 0.047,Y -402.513,Z 857.678,A 0.000,B 0.000,C 90.000,E1 158.050} C_DIS
LIN {X 0.032,Y -413.264,Z 857.676,A 0.000,B 0.000,C 90.000,E1 157.614} C_DIS
LIN {X -0.135,Y -416.836,Z 857.675,A 0.000,B 0.000,C 90.000,E1 157.486} C_DIS
LIN {X 0.045,Y -424.757,Z 857.673,A 0.000,B 0.000,C 90.000,E1 157.050} C_DIS
LIN {X -0.231,Y -432.974,Z 857.670,A 0.000,B 0.000,C 90.000,E1 156.613} C_DIS
LIN {X 0.173,Y -440.994,Z 857.667,A 0.000,B 0.000,C 90.000,E1 156.049} C_DIS
LIN {X 0.026,Y -445.635,Z 857.665,A 0.000,B 0.000,C 90.000,E1 155.741} C_DIS
LIN {X 0.157,Y -450.176,Z 857.663,A 0.000,B 0.000,C 90.000,E1 155.357} C_DIS
LIN {X 0.139,Y -457.803,Z 857.660,A 0.000,B 0.000,C 90.000,E1 154.717} C_DIS
LIN {X -0.110,Y -465.180,Z 857.656,A 0.000,B 0.000,C 90.000,E1 154.076} C_DIS
LIN {X -0.020,Y -470.873,Z 857.653,A 0.000,B 0.000,C 90.000,E1 153.512} C_DIS
LIN {X 0.102,Y -476.280,Z 857.650,A 0.000,B 0.000,C 90.000,E1 152.922} C_DIS
LIN {X 0.040,Y -480.171,Z 857.647,A 0.000,B 0.000,C 90.000,E1 152.487} C_DIS
LIN {X -0.217,Y -486.465,Z 857.643,A 0.000,B 0.000,C 90.000,E1 151.769} C_DIS
LIN {X -0.142,Y -496.254,Z 857.636,A 0.000,B 0.000,C 90.000,E1 150.539} C_DIS
LIN {X 0.062,Y -500.806,Z 857.633,A 0.000,B 0.000,C 90.000,E1 149.921} C_DIS
LIN {X 0.076,Y -510.774,Z 857.626,A 0.000,B 0.000,C 90.000,E1 148.584} C_DIS
LIN {X -0.087,Y -517.679,Z 857.620,A 0.000,B 0.000,C 90.000,E1 147.582} C_DIS
LIN {X -0.115,Y -523.139,Z 857.615,A 0.000,B 0.000,C 90.000,E1 146.707} C_DIS
LIN {X -0.154,Y -525.046,Z 857.613,A 0.000,B 0.000,C 90.000,E1 146.421} C_DIS
LIN {X -0.001,Y -532.472,Z 857.606,A 0.000,B 0.000,C 90.000,E1 145.102} C_DIS
LIN {X -0.015,Y -537.100,Z 857.601,A 0.000,B 0.000,C 90.000,E1 144.242} C_DIS
LIN {X -0.176,Y -547.883,Z 857.590,A 0.000,B 0.000,C 90.000,E1 142.271} C_DIS
LIN {X 0.246,Y -560.073,Z 857.578,A 0.000,B 0.000,C 90.000,E1 139.989} C_DIS
LIN {X -0.100,Y -565.265,Z 857.573,A 0.000,B 0.000,C 90.000,E1 139.057} C_DIS
LIN {X 0.041,Y -570.063,Z 857.567,A 0.000,B 0.000,C 90.000,E1 138.081} C_DIS
LIN {X -0.022,Y -574.251,Z 857.563,A 0.000,B 0.000,C 90.000,E1 137.268} C_DIS
LIN {X 0.064,Y -583.650,Z 857.552,A 0.000,B 0.000,C 90.000,E1 135.364} C_DIS
LIN {X 0.329,Y -590.784,Z 857.544,A 0.000,B 0.000,C 90.000,E1 133.866} C_DIS
LIN {X -0.106,Y -597.566,Z 857.536,A 0.000,B 0.000,C 90.000,E1 132.447} C_DIS
LIN {X -0.305,Y -603.385,Z 857.529,A 0.000,B 0.000,C 90.000,E1 131.148} C_DIS
LIN {X -0.212,Y -607.798,Z 857.523,A 0.000,B 0.000,C 90.000,E1 130.092} C_DIS
LIN {X -0.061,Y -611.919,Z 857.517,A 0.000,B 0.000,C 90.000,E1 129.036} C_DIS
LIN {X -0.242,Y -615.752,Z 857.511,A 0.000,B 0.000,C 90.000,E1 128.016} C_DIS
LIN {X 0.213,Y -621.963,Z 857.501,A 0.000,B 0.000,C 90.000,E1 126.171} C_DIS
LIN {X -0.201,Y -625.272,Z 857.495,A 0.000,B 0.000,C 90.000,E1 125.185} C_DIS
LIN {X 0.295,Y -628.229,Z 857.490,A 0.000,B 0.000,C 90.000,E1 124.119} C_DIS
LIN {X 0.119,Y -629.617,Z 857.487,A 0.000,B 0.000,C 90.000,E1 123.627} C_DIS
LIN {X 0.329,Y -632.568,Z 857.480,A 0.000,B 0.000,C 90.000,E1 122.339} C_DIS
LIN {X -0.161,Y -633.688,Z 857.477,A 0.000,B 0.000,C 90.000,E1 121.878} C_DIS
LIN {X 0.118,Y -636.124,Z 857.470,A 0.000,B 0.000,C 90.000,E1 120.590} C_DIS
LIN {X 0.108,Y -638.116,Z 857.463,A 0.000,B 0.000,C 90.000,E1 119.333} C_DIS
LIN {X -0.237,Y -639.601,Z 857.457,A 0.000,B 0.000,C 90.000,E1 118.359} C_DIS
LIN {X -0.056,Y -640.582,Z 857.453,A 0.000,B 0.000,C 90.000,E1 117.590} C_DIS
LIN {X 0.139,Y -641.310,Z 857.449,A 0.000,B 0.000,C 90.000,E1 116.821} C_DIS
LIN {X -0.167,Y -641.942,Z 857.444,A 0.000,B 0.000,C 90.000,E1 115.848} C_DIS
LIN {X 0.103,Y -642.157,Z 857.438,A 0.000,B 0.000,C 90.000,E1 114.823} C_DIS
LIN {X -0.098,Y -642.174,Z 857.437,A 0.000,B 0.000,C 90.000,E1 114.591} C_DIS
LIN {X 0.102,Y -641.439,Z 857.432,A 0.000,B 0.000,C 90.000,E1 113.823} C_DIS
LIN {X -0.026,Y -640.300,Z 857.430,A 0.000,B 0.000,C 90.000,E1 113.334} C_DIS
LIN {X 0.090,Y -638.009,Z 857.427,A 0.000,B 0.000,C 90.000,E1 112.823} C_DIS
LIN {X -0.102,Y -636.329,Z 857.425,A 0.000,B 0.000,C 90.000,E1 112.589} C_DIS
LIN {X -0.057,Y -634.252,Z 857.424,A 0.000,B 0.000,C 90.000,E1 112.333} C_DIS
LIN {X -0.038,Y -633.027,Z 857.423,A 0.000,B 0.000,C 90.000,E1 112.206} C_DIS
LIN {X -0.129,Y -627.081,Z 857.421,A 0.000,B 0.000,C 90.000,E1 111.716} C_DIS
LIN {X 0.057,Y -620.607,Z 857.418,A 0.000,B 0.000,C 90.000,E1 111.280} C_DIS
LIN {X 0.058,Y -609.036,Z 857.415,A 0.000,B 0.000,C 90.000,E1 110.663} C_DIS
LIN {X 0.122,Y -597.677,Z 857.412,A 0.000,B 0.000,C 90.000,E1 110.066} C_DIS
LIN {X -0.136,Y -589.183,Z 857.409,A 0.000,B 0.000,C 90.000,E1 109.685} C_DIS
LIN {X -0.092,Y -582.066,Z 857.408,A 0.000,B 0.000,C 90.000,E1 109.396} C_DIS
LIN {X 0.070,Y -572.686,Z 857.406,A 0.000,B 0.000,C 90.000,E1 109.087} C_DIS
LIN {X -0.246,Y -566.946,Z 857.405,A 0.000,B 0.000,C 90.000,E1 108.906} C_DIS
LIN {X 0.241,Y -565.497,Z 857.405,A 0.000,B 0.000,C 90.000,E1 108.779} C_DIS
LIN {X -0.243,Y -562.947,Z 857.403,A 0.000,B 0.000,C 90.000,E1 108.598} C_DIS
LIN {X 0.251,Y -562.932,Z 857.403,A 0.000,B 0.000,C 90.000,E1 108.544} C_DIS
LIN {X 0.109,Y -562.159,Z 857.402,A 0.000,B 0.000,C 90.000,E1 108.362} C_DIS
LIN {X -0.144,Y -561.116,Z 857.401,A 0.000,B 0.000,C 90.000,E1 108.181} C_DIS
LIN {X -0.172,Y -560.236,Z 857.399,A 0.000,B 0.000,C 90.000,E1 107.764} C_DIS
LIN {X -0.269,Y -559.825,Z 857.396,A 0.000,B 0.000,C 90.000,E1 107.221} C_DIS
LIN {X 0.059,Y -561.034,Z 857.369,A 0.000,B 0.000,C 90.000,E1 102.479} C_DIS
LIN {X 0.197,Y -562.465,Z 857.357,A 0.000,B 0.000,C 90.000,E1 100.254} C_DIS
LIN {X -0.061,Y -563.644,Z 857.348,A 0.000,B 0.000,C 90.000,E1 98.624} C_DIS
LIN {X -0.145,Y -564.410,Z 857.342,A 0.000,B 0.000,C 90.000,E1 97.530} C_DIS
LIN {X 0.106,Y -565.348,Z 857.333,A 0.000,B 0.000,C 90.000,E1 95.853} C_DIS
LIN {X 0.261,Y -566.107,Z 857.323,A 0.000,B 0.000,C 90.000,E1 94.188} C_DIS
LIN {X 0.208,Y -566.538,Z 857.317,A 0.000,B 0.000,C 90.000,E1 93.094} C_DIS
LIN {X 0.237,Y -566.935,Z 857.310,A 0.000,B 0.000,C 90.000,E1 91.718} C_DIS
LIN {X -0.187,Y -567.392,Z 857.301,A 0.000,B 0.000,C 90.000,E1 90.115} C_DIS
LIN {X 0.105,Y -567.815,Z 857.290,A 0.000,B 0.000,C 90.000,E1 88.165} C_DIS
LIN {X 0.167,Y -568.051,Z 857.282,A 0.000,B 0.000,C 90.000,E1 86.788} C_DIS
LIN {X -0.181,Y -568.342,Z 857.273,A 0.000,B 0.000,C 90.000,E1 85.179} C_DIS
LIN {X 0.200,Y -568.686,Z 857.263,A 0.000,B 0.000,C 90.000,E1 83.223} C_DIS
LIN {X -0.125,Y -569.317,Z 857.249,A 0.000,B 0.000,C 90.000,E1 80.792} C_DIS
LIN {X 0.134,Y -570.108,Z 857.237,A 0.000,B 0.000,C 90.000,E1 78.578} C_DIS
LIN {X 0.148,Y -570.742,Z 857.228,A 0.000,B 0.000,C 90.000,E1 76.937} C_DIS
LIN {X -0.213,Y -571.148,Z 857.221,A 0.000,B 0.000,C 90.000,E1 75.880} C_DIS
LIN {X 0.094,Y -571.528,Z 857.212,A 0.000,B 0.000,C 90.000,E1 74.212} C_DIS
LIN {X -0.114,Y -571.764,Z 857.206,A 0.000,B 0.000,C 90.000,E1 73.142} C_DIS
LIN {X -0.170,Y -571.942,Z 857.197,A 0.000,B 0.000,C 90.000,E1 71.511} C_DIS
LIN {X -0.246,Y -571.930,Z 857.185,A 0.000,B 0.000,C 90.000,E1 69.337} C_DIS
LIN {X -0.078,Y -571.849,Z 857.174,A 0.000,B 0.000,C 90.000,E1 67.411} C_DIS
LIN {X -0.097,Y -571.760,Z 857.167,A 0.000,B 0.000,C 90.000,E1 66.049} C_DIS
LIN {X -0.059,Y -571.405,Z 857.158,A 0.000,B 0.000,C 90.000,E1 64.409} C_DIS
LIN {X -0.122,Y -571.017,Z 857.150,A 0.000,B 0.000,C 90.000,E1 63.050} C_DIS
LIN {X -0.285,Y -570.691,Z 857.144,A 0.000,B 0.000,C 90.000,E1 61.975} C_DIS
LIN {X 0.082,Y -570.166,Z 857.138,A 0.000,B 0.000,C 90.000,E1 60.845} C_DIS
LIN {X 0.164,Y -569.606,Z 857.132,A 0.000,B 0.000,C 90.000,E1 59.744} C_DIS
LIN {X -0.153,Y -568.456,Z 857.124,A 0.000,B 0.000,C 90.000,E1 58.408} C_DIS
LIN {X 0.005,Y -567.462,Z 857.118,A 0.000,B 0.000,C 90.000,E1 57.296} C_DIS
LIN {X -0.269,Y -566.520,Z 857.114,A 0.000,B 0.000,C 90.000,E1 56.501} C_DIS
LIN {X -0.134,Y -565.071,Z 857.108,A 0.000,B 0.000,C 90.000,E1 55.388} C_DIS
LIN {X -0.127,Y -563.872,Z 857.103,A 0.000,B 0.000,C 90.000,E1 54.562} C_DIS
LIN {X 0.192,Y -562.573,Z 857.099,A 0.000,B 0.000,C 90.000,E1 53.703} C_DIS
LIN {X -0.189,Y -560.541,Z 857.092,A 0.000,B 0.000,C 90.000,E1 52.637} C_DIS
LIN {X 0.092,Y -558.825,Z 857.088,A 0.000,B 0.000,C 90.000,E1 51.778} C_DIS
LIN {X -0.085,Y -556.890,Z 857.083,A 0.000,B 0.000,C 90.000,E1 50.964} C_DIS
LIN {X -0.356,Y -555.475,Z 857.080,A 0.000,B 0.000,C 90.000,E1 50.436} C_DIS
LIN {X 0.216,Y -553.010,Z 857.075,A 0.000,B 0.000,C 90.000,E1 49.542} C_DIS
LIN {X -0.024,Y -550.244,Z 857.071,A 0.000,B 0.000,C 90.000,E1 48.728} C_DIS
LIN {X 0.068,Y -547.082,Z 857.066,A 0.000,B 0.000,C 90.000,E1 47.877} C_DIS
LIN {X 0.126,Y -543.622,Z 857.061,A 0.000,B 0.000,C 90.000,E1 47.025} C_DIS
LIN {X -0.056,Y -541.730,Z 857.059,A 0.000,B 0.000,C 90.000,E1 46.620} C_DIS
LIN {X 0.127,Y -538.338,Z 857.055,A 0.000,B 0.000,C 90.000,E1 45.891} C_DIS
LIN {X -0.083,Y -536.248,Z 857.053,A 0.000,B 0.000,C 90.000,E1 45.486} C_DIS
LIN {X 0.051,Y -532.192,Z 857.049,A 0.000,B 0.000,C 90.000,E1 44.757} C_DIS
LIN {X -0.019,Y -528.705,Z 857.046,A 0.000,B 0.000,C 90.000,E1 44.190} C_DIS
LIN {X 0.041,Y -523.859,Z 857.042,A 0.000,B 0.000,C 90.000,E1 43.461} C_DIS
LIN {X 0.141,Y -520.821,Z 857.039,A 0.000,B 0.000,C 90.000,E1 43.014} C_DIS
LIN {X -0.015,Y -516.465,Z 857.036,A 0.000,B 0.000,C 90.000,E1 42.447} C_DIS
LIN {X 0.304,Y -510.601,Z 857.032,A 0.000,B 0.000,C 90.000,E1 41.676} C_DIS
LIN {X -0.249,Y -505.572,Z 857.029,A 0.000,B 0.000,C 90.000,E1 41.148} C_DIS
LIN {X 0.108,Y -498.839,Z 857.024,A 0.000,B 0.000,C 90.000,E1 40.378} C_DIS
LIN {X 0.136,Y -493.251,Z 857.021,A 0.000,B 0.000,C 90.000,E1 39.806} C_DIS
LIN {X 0.061,Y -488.959,Z 857.019,A 0.000,B 0.000,C 90.000,E1 39.402} C_DIS
LIN {X -0.132,Y -480.184,Z 857.015,A 0.000,B 0.000,C 90.000,E1 38.624} C_DIS
LIN {X -0.065,Y -469.514,Z 857.010,A 0.000,B 0.000,C 90.000,E1 37.729} C_DIS
LIN {X 0.199,Y -461.717,Z 857.006,A 0.000,B 0.000,C 90.000,E1 37.076} C_DIS
LIN {X -0.065,Y -449.160,Z 857.001,A 0.000,B 0.000,C 90.000,E1 36.137} C_DIS
LIN {X 0.079,Y -435.029,Z 856.995,A 0.000,B 0.000,C 90.000,E1 35.025} C_DIS
LIN {X 0.032,Y -416.477,Z 856.986,A 0.000,B 0.000,C 90.000,E1 33.499} C_DIS
LIN {X -0.025,Y -404.609,Z 856.980,A 0.000,B 0.000,C 90.000,E1 32.418} C_DIS
LIN {X -0.091,Y -401.642,Z 856.979,A 0.000,B 0.000,C 90.000,E1 32.133} C_DIS
LIN {X 0.147,Y -397.874,Z 856.976,A 0.000,B 0.000,C 90.000,E1 31.671} C_DIS
LIN {X 0.169,Y -394.051,Z 856.973,A 0.000,B 0.000,C 90.000,E1 31.131} C_DIS
LIN {X -0.135,Y -392.000,Z 856.971,A 0.000,B 0.000,C 90.000,E1 30.718} C_DIS
LIN {X -0.010,Y -390.541,Z 856.967,A 0.000,B 0.000,C 90.000,E1 30.079} C_DIS
LIN {X 0.225,Y -390.033,Z 856.963,A 0.000,B 0.000,C 90.000,E1 29.333} C_DIS
LIN {X -0.080,Y -389.909,Z 856.959,A 0.000,B 0.000,C 90.000,E1 28.665} C_DIS
LIN {X 0.098,Y -392.002,Z 856.939,A 0.000,B 0.000,C 90.000,E1 25.079} C_DIS
LIN {X 0.095,Y -393.698,Z 856.928,A 0.000,B 0.000,C 90.000,E1 22.950} C_DIS
LIN {X 0.103,Y -396.346,Z 856.912,A 0.000,B 0.000,C 90.000,E1 20.120} C_DIS
LIN {X -0.119,Y -399.740,Z 856.894,A 0.000,B 0.000,C 90.000,E1 16.985} C_DIS
LIN {X -0.136,Y -402.801,Z 856.881,A 0.000,B 0.000,C 90.000,E1 14.537} C_DIS
LIN {X 0.119,Y -406.254,Z 856.867,A 0.000,B 0.000,C 90.000,E1 12.063} C_DIS
LIN {X -0.119,Y -409.523,Z 856.856,A 0.000,B 0.000,C 90.000,E1 10.018} C_DIS
LIN {X -0.010,Y -412.922,Z 856.844,A 0.000,B 0.000,C 90.000,E1 7.936} C_DIS
LIN {X 0.192,Y -417.186,Z 856.831,A 0.000,B 0.000,C 90.000,E1 5.511} C_DIS
LIN {X 0.158,Y -423.774,Z 856.812,A 0.000,B 0.000,C 90.000,E1 2.121} C_DIS
LIN {X -0.198,Y -429.761,Z 856.797,A 0.000,B 0.000,C 90.000,E1 359.484} C_DIS
LIN {X 0.047,Y -436.191,Z 856.782,A 0.000,B 0.000,C 90.000,E1 356.788} C_DIS
LIN {X -0.193,Y -444.086,Z 856.766,A 0.000,B 0.000,C 90.000,E1 353.856} C_DIS
LIN {X 0.029,Y -445.889,Z 856.763,A 0.000,B 0.000,C 90.000,E1 353.337} C_DIS
LIN {X -0.034,Y -447.247,Z 856.761,A 0.000,B 0.000,C 90.000,E1 353.053} C_DIS
LIN {X -0.204,Y -450.470,Z 856.759,A 0.000,B 0.000,C 90.000,E1 352.648} C_DIS
LIN {X -0.082,Y -451.572,Z 856.758,A 0.000,B 0.000,C 90.000,E1 352.470} C_DIS
LIN {X 0.005,Y -457.577,Z 856.756,A 0.000,B 0.000,C 90.000,E1 352.008} C_DIS
LIN {X 0.214,Y -477.019,Z 856.750,A 0.000,B 0.000,C 90.000,E1 351.027} C_DIS
LIN {X -0.166,Y -488.264,Z 856.747,A 0.000,B 0.000,C 90.000,E1 350.443} C_DIS
LIN {X -0.187,Y -497.988,Z 856.744,A 0.000,B 0.000,C 90.000,E1 349.859} C_DIS
LIN {X 0.133,Y -510.602,Z 856.739,A 0.000,B 0.000,C 90.000,E1 348.993} C_DIS
LIN {X 0.276,Y -519.932,Z 856.735,A 0.000,B 0.000,C 90.000,E1 348.342} C_DIS
LIN {X 0.085,Y -529.045,Z 856.732,A 0.000,B 0.000,C 90.000,E1 347.701} C_DIS
LIN {X 0.193,Y -540.788,Z 856.727,A 0.000,B 0.000,C 90.000,E1 346.756} C_DIS
LIN {X 0.045,Y -547.816,Z 856.723,A 0.000,B 0.000,C 90.000,E1 346.172} C_DIS
LIN {X 0.295,Y -554.545,Z 856.720,A 0.000,B 0.000,C 90.000,E1 345.519} C_DIS
LIN {X -0.159,Y -561.118,Z 856.716,A 0.000,B 0.000,C 90.000,E1 344.921} C_DIS
LIN {X -0.221,Y -566.133,Z 856.713,A 0.000,B 0.000,C 90.000,E1 344.393} C_DIS
LIN {X 0.014,Y -572.192,Z 856.709,A 0.000,B 0.000,C 90.000,E1 343.685} C_DIS
LIN {X 0.092,Y -575.607,Z 856.707,A 0.000,B 0.000,C 90.000,E1 343.268} C_DIS
LIN {X -0.253,Y -582.023,Z 856.703,A 0.000,B 0.000,C 90.000,E1 342.489} C_DIS
LIN {X -0.279,Y -587.052,Z 856.699,A 0.000,B 0.000,C 90.000,E1 341.819} C_DIS
LIN {X 0.301,Y -591.590,Z 856.695,A 0.000,B 0.000,C 90.000,E1 341.094} C_DIS
LIN {X 0.058,Y -597.533,Z 856.690,A 0.000,B 0.000,C 90.000,E1 340.188} C_DIS
LIN {X 0.130,Y -602.288,Z 856.686,A 0.000,B 0.000,C 90.000,E1 339.390} C_DIS
LIN {X -0.064,Y -608.995,Z 856.679,A 0.000,B 0.000,C 90.000,E1 338.230} C_DIS
LIN {X 0.103,Y -613.981,Z 856.674,A 0.000,B 0.000,C 90.000,E1 337.305} C_DIS
LIN {X 0.006,Y -618.687,Z 856.669,A 0.000,B 0.000,C 90.000,E1 336.410} C_DIS
LIN {X 0.291,Y -623.165,Z 856.664,A 0.000,B 0.000,C 90.000,E1 335.485} C_DIS
LIN {X 0.056,Y -628.453,Z 856.658,A 0.000,B 0.000,C 90.000,E1 334.357} C_DIS
LIN {X 0.095,Y -630.749,Z 856.655,A 0.000,B 0.000,C 90.000,E1 333.845} C_DIS
LIN {X -0.304,Y -635.908,Z 856.648,A 0.000,B 0.000,C 90.000,E1 332.615} C_DIS
LIN {X 0.193,Y -639.801,Z 856.642,A 0.000,B 0.000,C 90.000,E1 331.563} C_DIS
LIN {X -0.057,Y -644.412,Z 856.635,A 0.000,B 0.000,C 90.000,E1 330.333} C_DIS
LIN {X 0.002,Y -647.893,Z 856.630,A 0.000,B 0.000,C 90.000,E1 329.331} C_DIS
LIN {X 0.195,Y -651.855,Z 856.623,A 0.000,B 0.000,C 90.000,E1 328.074} C_DIS
LIN {X -0.206,Y -654.731,Z 856.617,A 0.000,B 0.000,C 90.000,E1 327.120} C_DIS
LIN {X -0.206,Y -657.456,Z 856.612,A 0.000,B 0.000,C 90.000,E1 326.135} C_DIS
LIN {X -0.061,Y -660.454,Z 856.605,A 0.000,B 0.000,C 90.000,E1 324.895} C_DIS
LIN {X -0.416,Y -663.103,Z 856.598,A 0.000,B 0.000,C 90.000,E1 323.703} C_DIS
LIN {X -0.338,Y -665.427,Z 856.591,A 0.000,B 0.000,C 90.000,E1 322.477} C_DIS
LIN {X -0.224,Y -667.284,Z 856.585,A 0.000,B 0.000,C 90.000,E1 321.251} C_DIS
LIN {X -0.164,Y -668.424,Z 856.581,A 0.000,B 0.000,C 90.000,E1 320.517} C_DIS
LIN {X 0.417,Y -670.439,Z 856.571,A 0.000,B 0.000,C 90.000,E1 318.771} C_DIS
LIN {X 0.127,Y -673.094,Z 856.559,A 0.000,B 0.000,C 90.000,E1 316.620} C_DIS
LIN {X 0.240,Y -674.622,Z 856.552,A 0.000,B 0.000,C 90.000,E1 315.405} C_DIS
LIN {X 0.293,Y -674.986,Z 856.550,A 0.000,B 0.000,C 90.000,E1 314.919} C_DIS
LIN {X 0.321,Y -675.326,Z 856.548,A 0.000,B 0.000,C 90.000,E1 314.676} C_DIS
LIN {X 0.070,Y -676.977,Z 856.539,A 0.000,B 0.000,C 90.000,E1 313.014} C_DIS
LIN {X -0.189,Y -678.415,Z 856.531,A 0.000,B 0.000,C 90.000,E1 311.595} C_DIS
LIN {X -0.367,Y -679.773,Z 856.523,A 0.000,B 0.000,C 90.000,E1 310.172} C_DIS
LIN {X -0.120,Y -680.800,Z 856.516,A 0.000,B 0.000,C 90.000,E1 308.955} C_DIS
LIN {X -0.124,Y -682.232,Z 856.507,A 0.000,B 0.000,C 90.000,E1 307.282} C_DIS
LIN {X -0.126,Y -683.370,Z 856.499,A 0.000,B 0.000,C 90.000,E1 305.851} C_DIS
LIN {X -0.129,Y -684.203,Z 856.493,A 0.000,B 0.000,C 90.000,E1 304.659} C_DIS
LIN {X 0.069,Y -685.175,Z 856.485,A 0.000,B 0.000,C 90.000,E1 303.214} C_DIS
LIN {X -0.031,Y -686.755,Z 856.473,A 0.000,B 0.000,C 90.000,E1 301.082} C_DIS
LIN {X -0.073,Y -688.434,Z 856.461,A 0.000,B 0.000,C 90.000,E1 298.949} C_DIS
LIN {X 0.095,Y -689.750,Z 856.453,A 0.000,B 0.000,C 90.000,E1 297.513} C_DIS
LIN {X -0.176,Y -691.622,Z 856.442,A 0.000,B 0.000,C 90.000,E1 295.643} C_DIS
LIN {X -0.138,Y -692.512,Z 856.437,A 0.000,B 0.000,C 90.000,E1 294.695} C_DIS
LIN {X 0.302,Y -693.022,Z 856.433,A 0.000,B 0.000,C 90.000,E1 293.951} C_DIS
LIN {X -0.127,Y -693.042,Z 856.431,A 0.000,B 0.000,C 90.000,E1 293.515} C_DIS
LIN {X 0.114,Y -693.005,Z 856.429,A 0.000,B 0.000,C 90.000,E1 293.259} C_DIS
LIN {X 0.083,Y -692.553,Z 856.428,A 0.000,B 0.000,C 90.000,E1 293.025} C_DIS
LIN {X -0.343,Y -691.172,Z 856.425,A 0.000,B 0.000,C 90.000,E1 292.589} C_DIS
LIN {X -0.225,Y -690.554,Z 856.425,A 0.000,B 0.000,C 90.000,E1 292.461} C_DIS
LIN {X 0.005,Y -688.706,Z 856.423,A 0.000,B 0.000,C 90.000,E1 292.206} C_DIS
LIN {X 0.083,Y -685.331,Z 856.421,A 0.000,B 0.000,C 90.000,E1 291.844} C_DIS
LIN {X 0.189,Y -683.641,Z 856.421,A 0.000,B 0.000,C 90.000,E1 291.716} C_DIS
LIN {X 0.038,Y -679.307,Z 856.420,A 0.000,B 0.000,C 90.000,E1 291.535} C_DIS
LIN {X -0.189,Y -674.030,Z 856.419,A 0.000,B 0.000,C 90.000,E1 291.354} C_DIS
LIN {X -0.206,Y -669.814,Z 856.418,A 0.000,B 0.000,C 90.000,E1 291.227} C_DIS
LIN {X 0.024,Y -654.783,Z 856.416,A 0.000,B 0.000,C 90.000,E1 290.865} C_DIS
LIN {X 0.109,Y -649.851,Z 856.415,A 0.000,B 0.000,C 90.000,E1 290.684} C_DIS
LIN {X 0.293,Y -647.902,Z 856.415,A 0.000,B 0.000,C 90.000,E1 290.610} C_DIS
LIN {X -0.075,Y -643.100,Z 856.413,A 0.000,B 0.000,C 90.000,E1 290.375} C_DIS
LIN {X -0.139,Y -642.031,Z 856.412,A 0.000,B 0.000,C 90.000,E1 290.248} C_DIS
LIN {X -0.183,Y -642.018,Z 856.412,A 0.000,B 0.000,C 90.000,E1 290.248} C_DIS
LIN {X -0.252,Y -641.822,Z 856.411,A 0.000,B 0.000,C 90.000,E1 290.066} C_DIS
LIN {X -0.021,Y -643.559,Z 856.409,A 0.000,B 0.000,C 90.000,E1 289.577} C_DIS
LIN {X 0.278,Y -650.902,Z 856.401,A 0.000,B 0.000,C 90.000,E1 288.181} C_DIS
LIN {X 0.045,Y -653.899,Z 856.398,A 0.000,B 0.000,C 90.000,E1 287.583} C_DIS
LIN {X -0.127,Y -657.148,Z 856.394,A 0.000,B 0.000,C 90.000,E1 286.858} C_DIS
LIN {X 0.358,Y -659.945,Z 856.390,A 0.000,B 0.000,C 90.000,E1 286.079} C_DIS
LIN {X 0.153,Y -661.583,Z 856.387,A 0.000,B 0.000,C 90.000,E1 285.607} C_DIS
LIN {X -0.131,Y -663.563,Z 856.383,A 0.000,B 0.000,C 90.000,E1 284.898} C_DIS
LIN {X -0.142,Y -664.688,Z 856.380,A 0.000,B 0.000,C 90.000,E1 284.411} C_DIS
LIN {X 0.161,Y -666.224,Z 856.375,A 0.000,B 0.000,C 90.000,E1 283.411} C_DIS
LIN {X -0.002,Y -666.752,Z 856.372,A 0.000,B 0.000,C 90.000,E1 282.939} C_DIS
LIN {X -0.308,Y -667.116,Z 856.369,A 0.000,B 0.000,C 90.000,E1 282.479} C_DIS
LIN {X 0.110,Y -667.356,Z 856.365,A 0.000,B 0.000,C 90.000,E1 281.715} C_DIS
LIN {X 0.032,Y -667.366,Z 856.364,A 0.000,B 0.000,C 90.000,E1 281.478} C_DIS
LIN {X -0.128,Y -667.127,Z 856.361,A 0.000,B 0.000,C 90.000,E1 281.007} C_DIS
LIN {X 0.239,Y -666.694,Z 856.358,A 0.000,B 0.000,C 90.000,E1 280.489} C_DIS
LIN {X -0.131,Y -665.595,Z 856.354,A 0.000,B 0.000,C 90.000,E1 279.792} C_DIS
LIN {X -0.308,Y -664.534,Z 856.352,A 0.000,B 0.000,C 90.000,E1 279.321} C_DIS
LIN {X 0.054,Y -663.160,Z 856.349,A 0.000,B 0.000,C 90.000,E1 278.803} C_DIS
LIN {X -0.245,Y -661.363,Z 856.346,A 0.000,B 0.000,C 90.000,E1 278.341} C_DIS
LIN {X -0.010,Y -658.202,Z 856.342,A 0.000,B 0.000,C 90.000,E1 277.587} C_DIS
LIN {X -0.337,Y -655.584,Z 856.339,A 0.000,B 0.000,C 90.000,E1 277.125} C_DIS
LIN {X -0.066,Y -651.831,Z 856.336,A 0.000,B 0.000,C 90.000,E1 276.486} C_DIS
LIN {X 0.209,Y -648.335,Z 856.333,A 0.000,B 0.000,C 90.000,E1 275.967} C_DIS
LIN {X -0.248,Y -644.253,Z 856.331,A 0.000,B 0.000,C 90.000,E1 275.511} C_DIS
LIN {X -0.092,Y -638.228,Z 856.327,A 0.000,B 0.000,C 90.000,E1 274.878} C_DIS
LIN {X -0.225,Y -632.780,Z 856.324,A 0.000,B 0.000,C 90.000,E1 274.416} C_DIS
LIN {X -0.171,Y -628.325,Z 856.323,A 0.000,B 0.000,C 90.000,E1 274.073} C_DIS
LIN {X 0.067,Y -625.461,Z 856.321,A 0.000,B 0.000,C 90.000,E1 273.841} C_DIS
LIN {X 0.228,Y -617.770,Z 856.319,A 0.000,B 0.000,C 90.000,E1 273.326} C_DIS
LIN {X 0.012,Y -611.430,Z 856.317,A 0.000,B 0.000,C 90.000,E1 272.980} C_DIS
LIN {X 0.042,Y -604.525,Z 856.315,A 0.000,B 0.000,C 90.000,E1 272.636} C_DIS
LIN {X -0.198,Y -597.638,Z 856.313,A 0.000,B 0.000,C 90.000,E1 272.350} C_DIS
LIN {X -0.015,Y -592.010,Z 856.312,A 0.000,B 0.000,C 90.000,E1 272.121} C_DIS
LIN {X -0.037,Y -584.446,Z 856.311,A 0.000,B 0.000,C 90.000,E1 271.892} C_DIS
LIN {X -0.254,Y -578.472,Z 856.310,A 0.000,B 0.000,C 90.000,E1 271.776} C_DIS
LIN {X -0.202,Y -571.719,Z 856.309,A 0.000,B 0.000,C 90.000,E1 271.661} C_DIS
LIN {X -0.128,Y -566.353,Z 856.309,A 0.000,B 0.000,C 90.000,E1 271.604} C_DIS
LIN {X -0.091,Y -554.818,Z 856.309,A 0.000,B 0.000,C 90.000,E1 271.547} C_DIS
LIN {X -0.247,Y -552.719,Z 856.308,A 0.000,B 0.000,C 90.000,E1 271.547} C_DIS
LIN {X -0.253,Y -549.257,Z 856.308,A 0.000,B 0.000,C 90.000,E1 271.432} C_DIS
LIN {X 0.108,Y -548.470,Z 856.307,A 0.000,B 0.000,C 90.000,E1 271.318} C_DIS
LIN {X -0.050,Y -547.795,Z 856.306,A 0.000,B 0.000,C 90.000,E1 271.146} C_DIS
LIN {X 0.193,Y -546.848,Z 856.304,A 0.000,B 0.000,C 90.000,E1 270.688} C_DIS
LIN {X -0.163,Y -545.614,Z 856.298,A 0.000,B 0.000,C 90.000,E1 269.599} C_DIS
LIN {X 0.147,Y -543.799,Z 856.285,A 0.000,B 0.000,C 90.000,E1 267.306} C_DIS
LIN {X -0.165,Y -542.662,Z 856.276,A 0.000,B 0.000,C 90.000,E1 265.641} C_DIS
LIN {X 0.088,Y -541.479,Z 856.266,A 0.000,B 0.000,C 90.000,E1 263.913} C_DIS
LIN {X 0.172,Y -540.750,Z 856.262,A 0.000,B 0.000,C 90.000,E1 263.053} C_DIS
LIN {X -0.100,Y -539.196,Z 856.252,A 0.000,B 0.000,C 90.000,E1 261.376} C_DIS
LIN {X 0.172,Y -538.185,Z 856.246,A 0.000,B 0.000,C 90.000,E1 260.208} C_DIS
LIN {X -0.127,Y -536.813,Z 856.238,A 0.000,B 0.000,C 90.000,E1 258.814} C_DIS
LIN {X 0.055,Y -535.939,Z 856.233,A 0.000,B 0.000,C 90.000,E1 257.937} C_DIS
LIN {X -0.067,Y -534.348,Z 856.225,A 0.000,B 0.000,C 90.000,E1 256.520} C_DIS
LIN {X 0.047,Y -531.521,Z 856.212,A 0.000,B 0.000,C 90.000,E1 254.212} C_DIS
LIN {X 0.009,Y -529.517,Z 856.203,A 0.000,B 0.000,C 90.000,E1 252.489} C_DIS
LIN {X 0.064,Y -527.707,Z 856.195,A 0.000,B 0.000,C 90.000,E1 251.040} C_DIS
LIN {X 0.263,Y -525.789,Z 856.187,A 0.000,B 0.000,C 90.000,E1 249.571} C_DIS
LIN {X -0.227,Y -524.276,Z 856.180,A 0.000,B 0.000,C 90.000,E1 248.465} C_DIS
LIN {X 0.265,Y -521.693,Z 856.171,A 0.000,B 0.000,C 90.000,E1 246.666} C_DIS
LIN {X 0.066,Y -519.458,Z 856.162,A 0.000,B 0.000,C 90.000,E1 245.229} C_DIS
LIN {X -0.090,Y -517.630,Z 856.156,A 0.000,B 0.000,C 90.000,E1 244.076} C_DIS
LIN {X 0.068,Y -516.168,Z 856.151,A 0.000,B 0.000,C 90.000,E1 243.179} C_DIS
LIN {X -0.024,Y -512.565,Z 856.140,A 0.000,B 0.000,C 90.000,E1 241.129} C_DIS
LIN {X -0.131,Y -511.053,Z 856.135,A 0.000,B 0.000,C 90.000,E1 240.255} C_DIS
LIN {X 0.055,Y -507.695,Z 856.125,A 0.000,B 0.000,C 90.000,E1 238.456} C_DIS
LIN {X 0.115,Y -504.817,Z 856.117,A 0.000,B 0.000,C 90.000,E1 236.962} C_DIS
LIN {X -0.073,Y -502.977,Z 856.112,A 0.000,B 0.000,C 90.000,E1 236.087} C_DIS
LIN {X -0.004,Y -501.023,Z 856.107,A 0.000,B 0.000,C 90.000,E1 235.182} C_DIS
LIN {X -0.083,Y -498.209,Z 856.100,A 0.000,B 0.000,C 90.000,E1 233.989} C_DIS
LIN {X 0.062,Y -493.244,Z 856.088,A 0.000,B 0.000,C 90.000,E1 231.859} C_DIS
LIN {X -0.236,Y -488.909,Z 856.078,A 0.000,B 0.000,C 90.000,E1 230.070} C_DIS
LIN {X -0.303,Y -484.774,Z 856.068,A 0.000,B 0.000,C 90.000,E1 228.243} C_DIS
LIN {X 0.112,Y -479.321,Z 856.054,A 0.000,B 0.000,C 90.000,E1 225.729} C_DIS
LIN {X 0.135,Y -475.352,Z 856.044,A 0.000,B 0.000,C 90.000,E1 223.866} C_DIS
LIN {X 0.169,Y -470.649,Z 856.032,A 0.000,B 0.000,C 90.000,E1 221.676} C_DIS
LIN {X 0.052,Y -466.590,Z 856.021,A 0.000,B 0.000,C 90.000,E1 219.806} C_DIS
LIN {X 0.087,Y -463.280,Z 856.012,A 0.000,B 0.000,C 90.000,E1 218.222} C_DIS
LIN {X 0.238,Y -459.348,Z 856.002,A 0.000,B 0.000,C 90.000,E1 216.297} C_DIS
LIN {X -0.142,Y -453.810,Z 855.988,A 0.000,B 0.000,C 90.000,E1 213.785} C_DIS
LIN {X -0.025,Y -449.007,Z 855.975,A 0.000,B 0.000,C 90.000,E1 211.514} C_DIS
LIN {X 0.093,Y -443.511,Z 855.961,A 0.000,B 0.000,C 90.000,E1 208.899} C_DIS
LIN {X 0.138,Y -440.151,Z 855.952,A 0.000,B 0.000,C 90.000,E1 207.257} C_DIS
LIN {X -0.097,Y -436.754,Z 855.942,A 0.000,B 0.000,C 90.000,E1 205.643} C_DIS
LIN {X 0.022,Y -432.682,Z 855.931,A 0.000,B 0.000,C 90.000,E1 203.643} C_DIS
LIN {X -0.115,Y -428.654,Z 855.920,A 0.000,B 0.000,C 90.000,E1 201.663} C_DIS
LIN {X -0.146,Y -425.366,Z 855.911,A 0.000,B 0.000,C 90.000,E1 199.993} C_DIS
LIN {X 0.051,Y -421.442,Z 855.900,A 0.000,B 0.000,C 90.000,E1 197.946} C_DIS
LIN {X -0.011,Y -418.226,Z 855.890,A 0.000,B 0.000,C 90.000,E1 196.260} C_DIS
LIN {X -0.049,Y -416.110,Z 855.885,A 0.000,B 0.000,C 90.000,E1 195.245} C_DIS
LIN {X -0.044,Y -412.553,Z 855.875,A 0.000,B 0.000,C 90.000,E1 193.536} C_DIS
LIN {X -0.022,Y -406.568,Z 855.858,A 0.000,B 0.000,C 90.000,E1 190.433} C_DIS
LIN {X 0.097,Y -403.127,Z 855.848,A 0.000,B 0.000,C 90.000,E1 188.681} C_DIS
LIN {X -0.046,Y -399.061,Z 855.837,A 0.000,B 0.000,C 90.000,E1 186.606} C_DIS
LIN {X -0.120,Y -392.937,Z 855.817,A 0.000,B 0.000,C 90.000,E1 183.094} C_DIS
LIN {X 0.031,Y -388.857,Z 855.801,A 0.000,B 0.000,C 90.000,E1 180.229} C_DIS
LIN {X -0.042,Y -386.408,Z 855.791,A 0.000,B 0.000,C 90.000,E1 178.453} C_DIS
LIN {X 0.045,Y -382.902,Z 855.777,A 0.000,B 0.000,C 90.000,E1 175.927} C_DIS
LIN {X 0.007,Y -380.902,Z 855.769,A 0.000,B 0.000,C 90.000,E1 174.489} C_DIS
LIN {X 0.013,Y -377.703,Z 855.755,A 0.000,B 0.000,C 90.000,E1 171.951} C_DIS
LIN {X 0.099,Y -373.029,Z 855.727,A 0.000,B 0.000,C 90.000,E1 166.825} C_DIS
LIN {X 0.131,Y -372.332,Z 855.719,A 0.000,B 0.000,C 90.000,E1 165.353} C_DIS
LIN {X -0.112,Y -372.188,Z 855.711,A 0.000,B 0.000,C 90.000,E1 163.921} C_DIS
LIN {X -0.146,Y -372.217,Z 855.709,A 0.000,B 0.000,C 90.000,E1 163.559} C_DIS
LIN {X 0.177,Y -372.424,Z 855.707,A 0.000,B 0.000,C 90.000,E1 163.142} C_DIS
LIN {X 0.145,Y -372.501,Z 855.705,A 0.000,B 0.000,C 90.000,E1 162.779} C_DIS
LIN {X 0.034,Y -373.609,Z 855.698,A 0.000,B 0.000,C 90.000,E1 161.710} C_DIS
LIN {X 0.052,Y -374.234,Z 855.696,A 0.000,B 0.000,C 90.000,E1 161.348} C_DIS
LIN {X 0.145,Y -374.704,Z 855.694,A 0.000,B 0.000,C 90.000,E1 160.967} C_DIS
LIN {X 0.100,Y -376.375,Z 855.690,A 0.000,B 0.000,C 90.000,E1 160.242} C_DIS
LIN {X 0.081,Y -377.505,Z 855.688,A 0.000,B 0.000,C 90.000,E1 159.880} C_DIS
LIN {X 0.065,Y -379.339,Z 855.686,A 0.000,B 0.000,C 90.000,E1 159.518} C_DIS
LIN {X 0.055,Y -381.221,Z 855.684,A 0.000,B 0.000,C 90.000,E1 159.156} C_DIS
LIN {X 0.191,Y -382.047,Z 855.683,A 0.000,B 0.000,C 90.000,E1 158.954} C_DIS
LIN {X 0.190,Y -383.264,Z 855.682,A 0.000,B 0.000,C 90.000,E1 158.773} C_DIS
LIN {X -0.162,Y -386.680,Z 855.680,A 0.000,B 0.000,C 90.000,E1 158.465} C_DIS
LIN {X 0.200,Y -389.726,Z 855.679,A 0.000,B 0.000,C 90.000,E1 158.156} C_DIS
LIN {X 0.018,Y -391.750,Z 855.678,A 0.000,B 0.000,C 90.000,E1 158.050} C_DIS
LIN {X 0.096,Y -397.733,Z 855.676,A 0.000,B 0.000,C 90.000,E1 157.720} C_DIS
LIN {X -0.061,Y -408.612,Z 855.674,A 0.000,B 0.000,C 90.000,E1 157.283} C_DIS
LIN {X 0.170,Y -415.527,Z 855.672,A 0.000,B 0.000,C 90.000,E1 156.975} C_DIS
LIN {X 0.184,Y -421.943,Z 855.671,A 0.000,B 0.000,C 90.000,E1 156.666} C_DIS
LIN {X -0.116,Y -428.611,Z 855.669,A 0.000,B 0.000,C 90.000,E1 156.357} C_DIS
LIN {X 0.082,Y -438.130,Z 855.665,A 0.000,B 0.000,C 90.000,E1 155.741} C_DIS
LIN {X -0.141,Y -446.022,Z 855.662,A 0.000,B 0.000,C 90.000,E1 155.229} C_DIS
LIN {X 0.125,Y -450.430,Z 855.660,A 0.000,B 0.000,C 90.000,E1 154.845} C_DIS
LIN {X 0.127,Y -459.322,Z 855.656,A 0.000,B 0.000,C 90.000,E1 154.101} C_DIS
LIN {X -0.059,Y -466.546,Z 855.653,A 0.000,B 0.000,C 90.000,E1 153.461} C_DIS
LIN {X 0.254,Y -471.967,Z 855.650,A 0.000,B 0.000,C 90.000,E1 152.871} C_DIS
LIN {X 0.103,Y -478.546,Z 855.645,A 0.000,B 0.000,C 90.000,E1 152.153} C_DIS
LIN {X 0.165,Y -485.152,Z 855.641,A 0.000,B 0.000,C 90.000,E1 151.385} C_DIS
LIN {X -0.205,Y -495.121,Z 855.634,A 0.000,B 0.000,C 90.000,E1 150.205} C_DIS
LIN {X -0.079,Y -507.727,Z 855.625,A 0.000,B 0.000,C 90.000,E1 148.535} C_DIS
LIN {X 0.141,Y -511.926,Z 855.622,A 0.000,B 0.000,C 90.000,E1 147.916} C_DIS
LIN {X 0.127,Y -517.751,Z 855.617,A 0.000,B 0.000,C 90.000,E1 147.041} C_DIS
LIN {X 0.113,Y -523.196,Z 855.612,A 0.000,B 0.000,C 90.000,E1 146.167} C_DIS
LIN {X -0.037,Y -529.915,Z 855.606,A 0.000,B 0.000,C 90.000,E1 145.022} C_DIS
LIN {X 0.204,Y -533.869,Z 855.602,A 0.000,B 0.000,C 90.000,E1 144.276} C_DIS
LIN {X 0.216,Y -539.955,Z 855.595,A 0.000,B 0.000,C 90.000,E1 143.130} C_DIS
LIN {X -0.298,Y -545.445,Z 855.590,A 0.000,B 0.000,C 90.000,E1 142.190} C_DIS
LIN {X 0.056,Y -557.840,Z 855.577,A 0.000,B 0.000,C 90.000,E1 139.908} C_DIS
LIN {X 0.106,Y -562.966,Z 855.572,A 0.000,B 0.000,C 90.000,E1 138.933} C_DIS
LIN {X 0.148,Y -570.058,Z 855.564,A 0.000,B 0.000,C 90.000,E1 137.553} C_DIS
LIN {X -0.204,Y -573.532,Z 855.561,A 0.000,B 0.000,C 90.000,E1 136.905} C_DIS
LIN {X 0.147,Y -579.600,Z 855.554,A 0.000,B 0.000,C 90.000,E1 135.648} C_DIS
LIN {X -0.078,Y -586.823,Z 855.546,A 0.000,B 0.000,C 90.000,E1 134.190} C_DIS
LIN {X 0.058,Y -592.494,Z 855.539,A 0.000,B 0.000,C 90.000,E1 132.975} C_DIS
LIN {X -0.076,Y -595.506,Z 855.535,A 0.000,B 0.000,C 90.000,E1 132.324} C_DIS
LIN {X 0.313,Y -600.185,Z 855.529,A 0.000,B 0.000,C 90.000,E1 131.229} C_DIS
LIN {X -0.094,Y -604.784,Z 855.523,A 0.000,B 0.000,C 90.000,E1 130.216} C_DIS
LIN {X -0.373,Y -608.930,Z 855.518,A 0.000,B 0.000,C 90.000,E1 129.197} C_DIS
LIN {X 0.267,Y -612.829,Z 855.512,A 0.000,B 0.000,C 90.000,E1 128.096} C_DIS
LIN {X 0.101,Y -616.347,Z 855.506,A 0.000,B 0.000,C 90.000,E1 127.076} C_DIS
LIN {X 0.160,Y -619.027,Z 855.502,A 0.000,B 0.000,C 90.000,E1 126.297} C_DIS
LIN {X -0.297,Y -622.193,Z 855.496,A 0.000,B 0.000,C 90.000,E1 125.311} C_DIS
LIN {X -0.199,Y -625.076,Z 855.490,A 0.000,B 0.000,C 90.000,E1 124.278} C_DIS
LIN {X -0.394,Y -626.478,Z 855.488,A 0.000,B 0.000,C 90.000,E1 123.785} C_DIS
LIN {X -0.239,Y -628.811,Z 855.482,A 0.000,B 0.000,C 90.000,E1 122.752} C_DIS
LIN {X 0.129,Y -630.447,Z 855.478,A 0.000,B 0.000,C 90.000,E1 121.957} C_DIS
LIN {X -0.185,Y -632.739,Z 855.471,A 0.000,B 0.000,C 90.000,E1 120.718} C_DIS
LIN {X -0.216,Y -635.237,Z 855.462,A 0.000,B 0.000,C 90.000,E1 119.205} C_DIS
LIN {X -0.084,Y -636.230,Z 855.458,A 0.000,B 0.000,C 90.000,E1 118.437} C_DIS
LIN {X -0.103,Y -637.600,Z 855.451,A 0.000,B 0.000,C 90.000,E1 117.180} C_DIS
LIN {X 0.054,Y -638.053,Z 855.447,A 0.000,B 0.000,C 90.000,E1 116.411} C_DIS
LIN {X -0.003,Y -638.300,Z 855.441,A 0.000,B 0.000,C 90.000,E1 115.412} C_DIS
LIN {X 0.162,Y -638.101,Z 855.437,A 0.000,B 0.000,C 90.000,E1 114.643} C_DIS
LIN {X 0.008,Y -637.667,Z 855.434,A 0.000,B 0.000,C 90.000,E1 114.155} C_DIS
LIN {X 0.111,Y -637.057,Z 855.431,A 0.000,B 0.000,C 90.000,E1 113.643} C_DIS
LIN {X 0.160,Y -636.340,Z 855.430,A 0.000,B 0.000,C 90.000,E1 113.387} C_DIS
LIN {X -0.043,Y -635.323,Z 855.429,A 0.000,B 0.000,C 90.000,E1 113.153} C_DIS
LIN {X 0.002,Y -634.150,Z 855.427,A 0.000,B 0.000,C 90.000,E1 112.898} C_DIS
LIN {X 0.073,Y -630.717,Z 855.424,A 0.000,B 0.000,C 90.000,E1 112.386} C_DIS
LIN {X -0.141,Y -627.675,Z 855.423,A 0.000,B 0.000,C 90.000,E1 112.153} C_DIS
LIN {X -0.158,Y -626.714,Z 855.422,A 0.000,B 0.000,C 90.000,E1 112.025} C_DIS
LIN {X -0.152,Y -625.578,Z 855.422,A 0.000,B 0.000,C 90.000,E1 111.897} C_DIS
LIN {X 0.196,Y -620.687,Z 855.420,A 0.000,B 0.000,C 90.000,E1 111.535} C_DIS
LIN {X 0.194,Y -619.103,Z 855.419,A 0.000,B 0.000,C 90.000,E1 111.408} C_DIS
LIN {X 0.175,Y -613.765,Z 855.417,A 0.000,B 0.000,C 90.000,E1 111.099} C_DIS
LIN {X 0.123,Y -610.796,Z 855.416,A 0.000,B 0.000,C 90.000,E1 110.918} C_DIS
LIN {X -0.107,Y -598.343,Z 855.412,A 0.000,B 0.000,C 90.000,E1 110.248} C_DIS
LIN {X 0.084,Y -589.983,Z 855.410,A 0.000,B 0.000,C 90.000,E1 109.812} C_DIS
LIN {X 0.047,Y -580.812,Z 855.408,A 0.000,B 0.000,C 90.000,E1 109.450} C_DIS
LIN {X 0.290,Y -571.698,Z 855.407,A 0.000,B 0.000,C 90.000,E1 109.141} C_DIS
LIN {X -0.237,Y -568.727,Z 855.406,A 0.000,B 0.000,C 90.000,E1 109.087} C_DIS
LIN {X -0.107,Y -566.151,Z 855.405,A 0.000,B 0.000,C 90.000,E1 108.960} C_DIS
LIN {X -0.111,Y -565.241,Z 855.405,A 0.000,B 0.000,C 90.000,E1 108.906} C_DIS
LIN {X 0.197,Y -563.667,Z 855.404,A 0.000,B 0.000,C 90.000,E1 108.725} C_DIS
LIN {X -0.206,Y -562.917,Z 855.404,A 0.000,B 0.000,C 90.000,E1 108.671} C_DIS
LIN {X -0.116,Y -561.693,Z 855.402,A 0.000,B 0.000,C 90.000,E1 108.308} C_DIS
LIN {X -0.226,Y -561.121,Z 855.401,A 0.000,B 0.000,C 90.000,E1 108.181} C_DIS
LIN {X 0.287,Y -560.314,Z 855.398,A 0.000,B 0.000,C 90.000,E1 107.692} C_DIS
LIN {X 0.155,Y -559.934,Z 855.393,A 0.000,B 0.000,C 90.000,E1 106.677} C_DIS
LIN {X -0.003,Y -560.608,Z 855.376,A 0.000,B 0.000,C 90.000,E1 103.647} C_DIS
LIN {X -0.039,Y -561.663,Z 855.365,A 0.000,B 0.000,C 90.000,E1 101.715} C_DIS
LIN {X -0.209,Y -562.810,Z 855.356,A 0.000,B 0.000,C 90.000,E1 100.074} C_DIS
LIN {X 0.004,Y -563.998,Z 855.347,A 0.000,B 0.000,C 90.000,E1 98.398} C_DIS
LIN {X 0.006,Y -564.720,Z 855.341,A 0.000,B 0.000,C 90.000,E1 97.296} C_DIS
LIN {X 0.198,Y -565.653,Z 855.331,A 0.000,B 0.000,C 90.000,E1 95.625} C_DIS
LIN {X -0.161,Y -566.401,Z 855.322,A 0.000,B 0.000,C 90.000,E1 94.012} C_DIS
LIN {X -0.248,Y -566.784,Z 855.316,A 0.000,B 0.000,C 90.000,E1 92.922} C_DIS
LIN {X -0.213,Y -567.182,Z 855.309,A 0.000,B 0.000,C 90.000,E1 91.547} C_DIS
LIN {X -0.184,Y -567.575,Z 855.301,A 0.000,B 0.000,C 90.000,E1 90.172} C_DIS
LIN {X 0.095,Y -568.009,Z 855.290,A 0.000,B 0.000,C 90.000,E1 88.224} C_DIS
LIN {X 0.147,Y -568.270,Z 855.283,A 0.000,B 0.000,C 90.000,E1 86.849} C_DIS
LIN {X -0.211,Y -568.523,Z 855.273,A 0.000,B 0.000,C 90.000,E1 85.241} C_DIS
LIN {X -0.235,Y -568.928,Z 855.261,A 0.000,B 0.000,C 90.000,E1 83.053} C_DIS
LIN {X -0.093,Y -569.493,Z 855.249,A 0.000,B 0.000,C 90.000,E1 80.849} C_DIS
LIN {X 0.175,Y -570.275,Z 855.237,A 0.000,B 0.000,C 90.000,E1 78.634} C_DIS
LIN {X 0.196,Y -570.905,Z 855.228,A 0.000,B 0.000,C 90.000,E1 76.992} C_DIS
LIN {X 0.028,Y -571.346,Z 855.220,A 0.000,B 0.000,C 90.000,E1 75.644} C_DIS
LIN {X -0.001,Y -571.665,Z 855.213,A 0.000,B 0.000,C 90.000,E1 74.283} C_DIS
LIN {X 0.131,Y -571.927,Z 855.205,A 0.000,B 0.000,C 90.000,E1 72.906} C_DIS
LIN {X 0.076,Y -572.079,Z 855.196,A 0.000,B 0.000,C 90.000,E1 71.275} C_DIS
LIN {X -0.161,Y -572.022,Z 855.185,A 0.000,B 0.000,C 90.000,E1 69.390} C_DIS
LIN {X -0.205,Y -571.923,Z 855.175,A 0.000,B 0.000,C 90.000,E1 67.486} C_DIS
LIN {X 0.003,Y -571.855,Z 855.167,A 0.000,B 0.000,C 90.000,E1 66.102} C_DIS
LIN {X 0.049,Y -571.455,Z 855.158,A 0.000,B 0.000,C 90.000,E1 64.460} C_DIS
LIN {X -0.266,Y -571.043,Z 855.151,A 0.000,B 0.000,C 90.000,E1 63.127} C_DIS
LIN {X 0.168,Y -570.575,Z 855.143,A 0.000,B 0.000,C 90.000,E1 61.719} C_DIS
LIN {X -0.243,Y -570.027,Z 855.137,A 0.000,B 0.000,C 90.000,E1 60.667} C_DIS
LIN {X 0.118,Y -569.391,Z 855.131,A 0.000,B 0.000,C 90.000,E1 59.537} C_DIS
LIN {X -0.200,Y -568.234,Z 855.123,A 0.000,B 0.000,C 90.000,E1 58.201} C_DIS
LIN {X -0.044,Y -567.106,Z 855.117,A 0.000,B 0.000,C 90.000,E1 57.089} C_DIS
LIN {X -0.322,Y -566.105,Z 855.113,A 0.000,B 0.000,C 90.000,E1 56.294} C_DIS
LIN {X -0.191,Y -564.624,Z 855.107,A 0.000,B 0.000,C 90.000,E1 55.182} C_DIS
LIN {X 0.137,Y -563.347,Z 855.102,A 0.000,B 0.000,C 90.000,E1 54.322} C_DIS
LIN {X 0.121,Y -561.977,Z 855.097,A 0.000,B 0.000,C 90.000,E1 53.497} C_DIS
LIN {X -0.026,Y -560.430,Z 855.093,A 0.000,B 0.000,C 90.000,E1 52.683} C_DIS
LIN {X 0.258,Y -558.698,Z 855.088,A 0.000,B 0.000,C 90.000,E1 51.823} C_DIS
LIN {X 0.083,Y -556.716,Z 855.083,A 0.000,B 0.000,C 90.000,E1 51.009} C_DIS
LIN {X -0.109,Y -554.462,Z 855.079,A 0.000,B 0.000,C 90.000,E1 50.194} C_DIS
LIN {X 0.030,Y -552.819,Z 855.076,A 0.000,B 0.000,C 90.000,E1 49.622} C_DIS
LIN {X 0.151,Y -550.032,Z 855.071,A 0.000,B 0.000,C 90.000,E1 48.771} C_DIS
LIN {X 0.245,Y -546.837,Z 855.066,A 0.000,B 0.000,C 90.000,E1 47.919} C_DIS
LIN {X -0.090,Y -544.574,Z 855.063,A 0.000,B 0.000,C 90.000,E1 47.391} C_DIS
LIN {X -0.070,Y -542.152,Z 855.060,A 0.000,B 0.000,C 90.000,E1 46.824} C_DIS
LIN {X -0.253,Y -538.736,Z 855.056,A 0.000,B 0.000,C 90.000,E1 46.134} C_DIS
LIN {X -0.277,Y -535.886,Z 855.053,A 0.000,B 0.000,C 90.000,E1 45.567} C_DIS
LIN {X -0.145,Y -531.785,Z 855.049,A 0.000,B 0.000,C 90.000,E1 44.838} C_DIS
LIN {X -0.217,Y -528.268,Z 855.046,A 0.000,B 0.000,C 90.000,E1 44.271} C_DIS
LIN {X 0.065,Y -524.399,Z 855.043,A 0.000,B 0.000,C 90.000,E1 43.662} C_DIS
LIN {X -0.061,Y -520.292,Z 855.039,A 0.000,B 0.000,C 90.000,E1 43.095} C_DIS
LIN {X -0.009,Y -517.053,Z 855.037,A 0.000,B 0.000,C 90.000,E1 42.651} C_DIS
LIN {X -0.025,Y -511.137,Z 855.033,A 0.000,B 0.000,C 90.000,E1 41.919} C_DIS
LIN {X 0.009,Y -507.429,Z 855.030,A 0.000,B 0.000,C 90.000,E1 41.472} C_DIS
LIN {X 0.056,Y -503.561,Z 855.028,A 0.000,B 0.000,C 90.000,E1 41.024} C_DIS
LIN {X 0.090,Y -496.701,Z 855.024,A 0.000,B 0.000,C 90.000,E1 40.297} C_DIS
LIN {X -0.114,Y -491.104,Z 855.021,A 0.000,B 0.000,C 90.000,E1 39.769} C_DIS
LIN {X -0.060,Y -484.097,Z 855.017,A 0.000,B 0.000,C 90.000,E1 39.116} C_DIS
LIN {X -0.090,Y -478.081,Z 855.014,A 0.000,B 0.000,C 90.000,E1 38.588} C_DIS
LIN {X 0.132,Y -468.956,Z 855.010,A 0.000,B 0.000,C 90.000,E1 37.810} C_DIS
LIN {X 0.055,Y -459.519,Z 855.006,A 0.000,B 0.000,C 90.000,E1 37.076} C_DIS
LIN {X -0.117,Y -445.414,Z 855.000,A 0.000,B 0.000,C 90.000,E1 36.011} C_DIS
LIN {X 0.116,Y -420.428,Z 854.989,A 0.000,B 0.000,C 90.000,E1 33.992} C_DIS
LIN {X -0.165,Y -404.001,Z 854.981,A 0.000,B 0.000,C 90.000,E1 32.546} C_DIS
LIN {X -0.187,Y -398.964,Z 854.978,A 0.000,B 0.000,C 90.000,E1 32.005} C_DIS
LIN {X -0.117,Y -396.387,Z 854.976,A 0.000,B 0.000,C 90.000,E1 31.671} C_DIS
LIN {X -0.072,Y -393.789,Z 854.974,A 0.000,B 0.000,C 90.000,E1 31.258} C_DIS
LIN {X -0.181,Y -392.272,Z 854.972,A 0.000,B 0.000,C 90.000,E1 30.924} C_DIS
LIN {X 0.017,Y -391.633,Z 854.971,A 0.000,B 0.000,C 90.000,E1 30.718} C_DIS
LIN {X 0.065,Y -390.334,Z 854.967,A 0.000,B 0.000,C 90.000,E1 30.001} C_DIS
LIN {X -0.046,Y -389.987,Z 854.962,A 0.000,B 0.000,C 90.000,E1 29.127} C_DIS
LIN {X 0.177,Y -390.259,Z 854.956,A 0.000,B 0.000,C 90.000,E1 28.025} C_DIS
LIN {X 0.138,Y -391.861,Z 854.942,A 0.000,B 0.000,C 90.000,E1 25.540} C_DIS
LIN {X -0.018,Y -393.797,Z 854.928,A 0.000,B 0.000,C 90.000,E1 23.078} C_DIS
LIN {X -0.005,Y -396.400,Z 854.913,A 0.000,B 0.000,C 90.000,E1 20.248} C_DIS
LIN {X -0.103,Y -399.758,Z 854.895,A 0.000,B 0.000,C 90.000,E1 17.094} C_DIS
LIN {X -0.055,Y -403.736,Z 854.877,A 0.000,B 0.000,C 90.000,E1 13.939} C_DIS
LIN {X 0.133,Y -407.294,Z 854.864,A 0.000,B 0.000,C 90.000,E1 11.478} C_DIS
LIN {X -0.081,Y -410.635,Z 854.852,A 0.000,B 0.000,C 90.000,E1 9.434} C_DIS
LIN {X 0.052,Y -414.083,Z 854.841,A 0.000,B 0.000,C 90.000,E1 7.352} C_DIS
LIN {X -0.192,Y -417.780,Z 854.830,A 0.000,B 0.000,C 90.000,E1 5.334} C_DIS
LIN {X -0.183,Y -425.142,Z 854.809,A 0.000,B 0.000,C 90.000,E1 1.604} C_DIS
LIN {X -0.127,Y -430.699,Z 854.795,A 0.000,B 0.000,C 90.000,E1 359.141} C_DIS
LIN {X 0.148,Y -437.187,Z 854.780,A 0.000,B 0.000,C 90.000,E1 356.445} C_DIS
LIN {X -0.182,Y -444.175,Z 854.766,A 0.000,B 0.000,C 90.000,E1 353.856} C_DIS
LIN {X 0.099,Y -446.509,Z 854.762,A 0.000,B 0.000,C 90.000,E1 353.166} C_DIS
LIN {X 0.160,Y -447.191,Z 854.761,A 0.000,B 0.000,C 90.000,E1 352.996} C_DIS
LIN {X 0.201,Y -449.533,Z 854.759,A 0.000,B 0.000,C 90.000,E1 352.648} C_DIS
LIN {X -0.123,Y -450.519,Z 854.758,A 0.000,B 0.000,C 90.000,E1 352.527} C_DIS
LIN {X -0.058,Y -451.804,Z 854.758,A 0.000,B 0.000,C 90.000,E1 352.356} C_DIS
LIN {X 0.111,Y -452.780,Z 854.757,A 0.000,B 0.000,C 90.000,E1 352.243} C_DIS
LIN {X -0.133,Y -457.039,Z 854.755,A 0.000,B 0.000,C 90.000,E1 351.951} C_DIS
LIN {X 0.003,Y -460.821,Z 854.754,A 0.000,B 0.000,C 90.000,E1 351.724} C_DIS
LIN {X -0.150,Y -477.544,Z 854.749,A 0.000,B 0.000,C 90.000,E1 350.905} C_DIS
LIN {X 0.114,Y -487.280,Z 854.746,A 0.000,B 0.000,C 90.000,E1 350.330} C_DIS
LIN {X 0.148,Y -496.911,Z 854.743,A 0.000,B 0.000,C 90.000,E1 349.746} C_DIS
LIN {X -0.072,Y -507.970,Z 854.739,A 0.000,B 0.000,C 90.000,E1 349.050} C_DIS
LIN {X -0.096,Y -514.242,Z 854.737,A 0.000,B 0.000,C 90.000,E1 348.634} C_DIS
LIN {X -0.152,Y -521.897,Z 854.734,A 0.000,B 0.000,C 90.000,E1 348.105} C_DIS
LIN {X 0.092,Y -529.467,Z 854.731,A 0.000,B 0.000,C 90.000,E1 347.521} C_DIS
LIN {X 0.194,Y -539.733,Z 854.726,A 0.000,B 0.000,C 90.000,E1 346.700} C_DIS
LIN {X 0.151,Y -544.028,Z 854.724,A 0.000,B 0.000,C 90.000,E1 346.353} C_DIS
LIN {X -0.028,Y -550.945,Z 854.721,A 0.000,B 0.000,C 90.000,E1 345.755} C_DIS
LIN {X -0.063,Y -559.004,Z 854.717,A 0.000,B 0.000,C 90.000,E1 344.991} C_DIS
LIN {X 0.094,Y -564.134,Z 854.714,A 0.000,B 0.000,C 90.000,E1 344.448} C_DIS
LIN {X 0.090,Y -571.468,Z 854.709,A 0.000,B 0.000,C 90.000,E1 343.630} C_DIS
LIN {X 0.064,Y -576.091,Z 854.706,A 0.000,B 0.000,C 90.000,E1 343.087} C_DIS
LIN {X 0.197,Y -583.533,Z 854.701,A 0.000,B 0.000,C 90.000,E1 342.127} C_DIS
LIN {X 0.260,Y -587.486,Z 854.698,A 0.000,B 0.000,C 90.000,E1 341.583} C_DIS
LIN {X 0.287,Y -592.020,Z 854.694,A 0.000,B 0.000,C 90.000,E1 340.913} C_DIS
LIN {X 0.049,Y -597.925,Z 854.689,A 0.000,B 0.000,C 90.000,E1 340.007} C_DIS
LIN {X 0.124,Y -602.717,Z 854.685,A 0.000,B 0.000,C 90.000,E1 339.209} C_DIS
LIN {X 0.161,Y -609.411,Z 854.678,A 0.000,B 0.000,C 90.000,E1 338.028} C_DIS
LIN {X 0.343,Y -614.386,Z 854.673,A 0.000,B 0.000,C 90.000,E1 337.102} C_DIS
LIN {X 0.020,Y -618.413,Z 854.669,A 0.000,B 0.000,C 90.000,E1 336.357} C_DIS
LIN {X -0.271,Y -622.917,Z 854.664,A 0.000,B 0.000,C 90.000,E1 335.485} C_DIS
LIN {X -0.246,Y -627.673,Z 854.658,A 0.000,B 0.000,C 90.000,E1 334.460} C_DIS
LIN {X -0.184,Y -631.120,Z 854.654,A 0.000,B 0.000,C 90.000,E1 333.691} C_DIS
LIN {X -0.003,Y -636.274,Z 854.647,A 0.000,B 0.000,C 90.000,E1 332.410} C_DIS
LIN {X 0.145,Y -639.197,Z 854.643,A 0.000,B 0.000,C 90.000,E1 331.641} C_DIS
LIN {X -0.118,Y -643.907,Z 854.636,A 0.000,B 0.000,C 90.000,E1 330.411} C_DIS
LIN {X 0.005,Y -648.290,Z 854.629,A 0.000,B 0.000,C 90.000,E1 329.154} C_DIS
LIN {X 0.109,Y -651.496,Z 854.623,A 0.000,B 0.000,C 90.000,E1 328.152} C_DIS
LIN {X 0.146,Y -655.126,Z 854.616,A 0.000,B 0.000,C 90.000,E1 326.914} C_DIS
LIN {X 0.155,Y -657.844,Z 854.611,A 0.000,B 0.000,C 90.000,E1 325.928} C_DIS
